ABB RAPID module: Template_20023_Module.mod

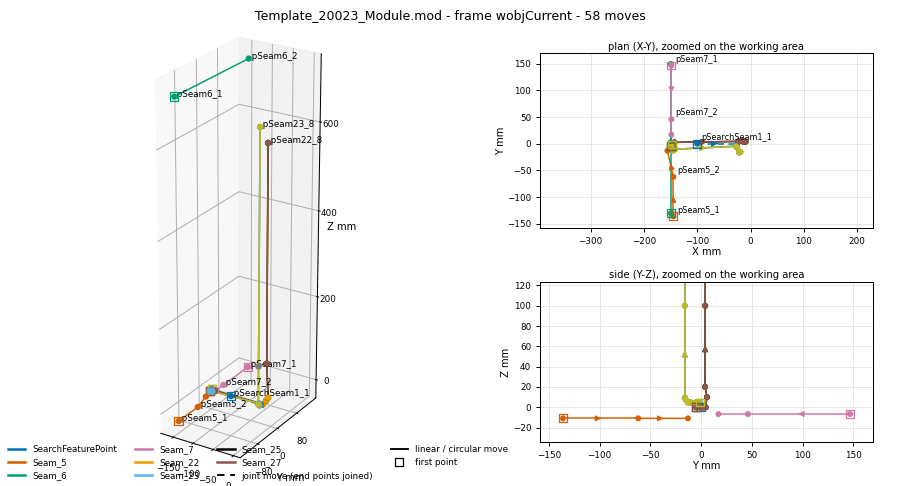
[picture p0: tool path of Template_20023_Module.mod in frame wobjCurrent, 58 of 171 moves have a stored position in this frame; points joined in program order, loops and branches not executed]
MODULE Template_20023_Module
    !*****************************************************
    !Module Name:   Template_20023_Module
    !Version:       1.0
    !Description:   All the targets are coordinated in its self coordinate system
    !Date:          2021-8-21
    !Author:        Michael
    !*****************************************************

    LOCAL PERS num numPartCount:=7;

    !For oframe searching
    LOCAL PERS robtarget pQ1_X1:=[[-75,0,0],[0.37941,0.915976,0.0499502,0.12059],[-1,-1,0,1],[-800,500,456,9E+9,9E+9,9E+9]];
    LOCAL PERS robtarget pQ1_X2:=[[-30,0,0],[0.37941,0.915976,0.0499502,0.12059],[-1,-1,0,1],[-800,500,456,9E+9,9E+9,9E+9]];
    LOCAL PERS robtarget pQ1_Y1:=[[0,75,0],[0.183013,-0.612372,0.683013,-0.353553],[-1,0,-1,1],[-800,500,456,9E+9,9E+9,9E+9]];
    LOCAL PERS robtarget pQ1_Y2:=[[0,200,0],[0.183013,-0.612372,0.683013,-0.353553],[-1,0,-1,1],[-800,500,456,9E+9,9E+9,9E+9]];
    LOCAL PERS robtarget pQ1_Z1:=[[0,0,50],[0.562422,0.303603,0.732963,-0.232963],[-1,-2,-1,1],[-800,500,456,9E+9,9E+9,9E+9]];
    LOCAL PERS robtarget pQ1_Z2:=[[0,0,250],[0.232963,0.732963,-0.303603,0.562422],[-2,-1,1,1],[-800,500,456,9E+9,9E+9,9E+9]];
    LOCAL PERS robtarget pQ1_X1_Found:=[[-75,0,0],[0.37941,0.915976,0.0499502,0.12059],[-1,-1,0,1],[-800,500,456,9E+9,9E+9,9E+9]];
    LOCAL PERS robtarget pQ1_X2_Found:=[[-30,0,0],[0.37941,0.915976,0.0499502,0.12059],[-1,-1,0,1],[-800,500,456,9E+9,9E+9,9E+9]];
    LOCAL PERS robtarget pQ1_Y1_Found:=[[0,75,0],[0.183013,-0.612372,0.683013,-0.353553],[-1,0,-1,1],[-800,500,456,9E+9,9E+9,9E+9]];
    LOCAL PERS robtarget pQ1_Y2_Found:=[[0,200,0],[0.183013,-0.612372,0.683013,-0.353553],[-1,0,-1,1],[-800,500,456,9E+9,9E+9,9E+9]];
    LOCAL PERS robtarget pQ1_Z1_Found:=[[0,0,50],[0.562422,0.303603,0.732963,-0.232963],[-1,-2,-1,1],[-800,500,456,9E+9,9E+9,9E+9]];
    LOCAL PERS robtarget pQ1_Z2_Found:=[[0,0,250],[0.232963,0.732963,-0.303603,0.562422],[-2,-1,1,1],[-800,500,456,9E+9,9E+9,9E+9]];

    LOCAL PERS robtarget pQ2_X1:=[[-75,0,0],[0.37941,0.915976,0.0499502,0.12059],[-1,-1,0,1],[-800,500,456,9E+9,9E+9,9E+9]];
    LOCAL PERS robtarget pQ2_X2:=[[-30,0,0],[0.37941,0.915976,0.0499502,0.12059],[-1,-1,0,1],[-800,500,456,9E+9,9E+9,9E+9]];
    LOCAL PERS robtarget pQ2_Y1:=[[-0.03,74.99,-0.03],[0.0903086,-0.672569,0.657682,-0.327031],[-1,-1,0,1],[-800,500,456.001,9E+09,9E+09,9E+09]];
    LOCAL PERS robtarget pQ2_Y2:=[[-0.03,200,-0.03],[0.0903092,-0.67257,0.657681,-0.327031],[-1,-1,0,1],[-800,500,456.001,9E+09,9E+09,9E+09]];
    LOCAL PERS robtarget pQ2_Z1:=[[0,0,50],[0.562422,0.303603,0.732963,-0.232963],[-1,-2,-1,1],[-800,500,456,9E+9,9E+9,9E+9]];
    LOCAL PERS robtarget pQ2_Z2:=[[0,0,250],[0.232963,0.732963,-0.303603,0.562422],[-2,-1,1,1],[-800,500,456,9E+9,9E+9,9E+9]];
    LOCAL PERS robtarget pQ2_X1_Found:=[[-75,0,0],[0.37941,0.915976,0.0499502,0.12059],[-1,-1,0,1],[-800,500,456,9E+9,9E+9,9E+9]];
    LOCAL PERS robtarget pQ2_X2_Found:=[[-30,0,0],[0.37941,0.915976,0.0499502,0.12059],[-1,-1,0,1],[-800,500,456,9E+9,9E+9,9E+9]];
    LOCAL PERS robtarget pQ2_Y1_Found:=[[17.85,90.22,0.26],[0.183013,-0.612372,0.683013,-0.353553],[-1,0,-1,1],[-800,500,456,9E+09,9E+09,9E+09]];
    LOCAL PERS robtarget pQ2_Y2_Found:=[[14.86,215.24,-0.11],[0.183013,-0.612372,0.683013,-0.353553],[-1,0,-1,1],[-800,500,456,9E+09,9E+09,9E+09]];
    LOCAL PERS robtarget pQ2_Z1_Found:=[[0,0,50],[0.562422,0.303603,0.732963,-0.232963],[-1,-2,-1,1],[-800,500,456,9E+9,9E+9,9E+9]];
    LOCAL PERS robtarget pQ2_Z2_Found:=[[16.02,7.07,231.87],[0.232963,0.732963,-0.303603,0.562422],[-2,-1,1,1],[-800,500,456,9E+09,9E+09,9E+09]];

    LOCAL PERS robtarget pQ3_X1:=[[-75,0,0],[0.37941,0.915976,0.0499502,0.12059],[-1,-1,0,1],[-800,500,456,9E+9,9E+9,9E+9]];
    LOCAL PERS robtarget pQ3_X2:=[[-30,0,0],[0.37941,0.915976,0.0499502,0.12059],[-1,-1,0,1],[-800,500,456,9E+9,9E+9,9E+9]];
    LOCAL PERS robtarget pQ3_Y1:=[[0,-300,0],[0.0890947,0.615873,0.708619,0.332599],[-2,0,-1,1],[-800,-500,450.515,9E+09,9E+09,9E+09]];
    LOCAL PERS robtarget pQ3_Y2:=[[0,-100,0],[0.0890967,0.615873,0.708619,0.332599],[-1,0,-2,1],[-800,-500,450.515,9E+09,9E+09,9E+09]];
    LOCAL PERS robtarget pQ3_Z1:=[[0,0,50],[0.562422,0.303603,0.732963,-0.232963],[-1,-2,-1,1],[-800,500,456,9E+9,9E+9,9E+9]];
    LOCAL PERS robtarget pQ3_Z2:=[[0,0,500],[0.326752,-0.683237,-0.28535,-0.587363],[-1,0,-1,1],[-800,-500,450.515,9E+09,9E+09,9E+09]];
    LOCAL PERS robtarget pQ3_X1_Found:=[[-75,0,0],[0.37941,0.915976,0.0499502,0.12059],[-1,-1,0,1],[-800,500,456,9E+9,9E+9,9E+9]];
    LOCAL PERS robtarget pQ3_X2_Found:=[[-30,0,0],[0.37941,0.915976,0.0499502,0.12059],[-1,-1,0,1],[-800,500,456,9E+9,9E+9,9E+9]];
    LOCAL PERS robtarget pQ3_Y1_Found:=[[5.33,-307.13,27.55],[0.183013,-0.612372,0.683013,-0.353553],[-1,0,-1,1],[-800,500,456,9E+09,9E+09,9E+09]];
    LOCAL PERS robtarget pQ3_Y2_Found:=[[4.1,-107.45,27.54],[0.183013,-0.612372,0.683013,-0.353553],[-1,0,-1,1],[-800,500,456,9E+09,9E+09,9E+09]];
    LOCAL PERS robtarget pQ3_Z1_Found:=[[0,0,50],[0.562422,0.303603,0.732963,-0.232963],[-1,-2,-1,1],[-800,500,456,9E+9,9E+9,9E+9]];
    LOCAL PERS robtarget pQ3_Z2_Found:=[[-3.2,-18.41,500.1],[0.232963,0.732963,-0.303603,0.562422],[-2,-1,1,1],[-800,500,456,9E+09,9E+09,9E+09]];

    LOCAL PERS robtarget pQ4_X1:=[[-75,0,0],[0.37941,0.915976,0.0499502,0.12059],[-1,-1,0,1],[-800,500,456,9E+9,9E+9,9E+9]];
    LOCAL PERS robtarget pQ4_X2:=[[-30,0,0],[0.37941,0.915976,0.0499502,0.12059],[-1,-1,0,1],[-800,500,456,9E+9,9E+9,9E+9]];
    LOCAL PERS robtarget pQ4_Y1:=[[0,75,0],[0.183013,-0.612372,0.683013,-0.353553],[-1,0,-1,1],[-800,500,456,9E+9,9E+9,9E+9]];
    LOCAL PERS robtarget pQ4_Y2:=[[0,200,0],[0.183013,-0.612372,0.683013,-0.353553],[-1,0,-1,1],[-800,500,456,9E+9,9E+9,9E+9]];
    LOCAL PERS robtarget pQ4_Z1:=[[0,0,50],[0.562422,0.303603,0.732963,-0.232963],[-1,-2,-1,1],[-800,500,456,9E+9,9E+9,9E+9]];
    LOCAL PERS robtarget pQ4_Z2:=[[0,0,250],[0.232963,0.732963,-0.303603,0.562422],[-2,-1,1,1],[-800,500,456,9E+9,9E+9,9E+9]];
    LOCAL PERS robtarget pQ4_X1_Found:=[[-75,0,0],[0.37941,0.915976,0.0499502,0.12059],[-1,-1,0,1],[-800,500,456,9E+9,9E+9,9E+9]];
    LOCAL PERS robtarget pQ4_X2_Found:=[[-30,0,0],[0.37941,0.915976,0.0499502,0.12059],[-1,-1,0,1],[-800,500,456,9E+9,9E+9,9E+9]];
    LOCAL PERS robtarget pQ4_Y1_Found:=[[0,75,0],[0.183013,-0.612372,0.683013,-0.353553],[-1,0,-1,1],[-800,500,456,9E+9,9E+9,9E+9]];
    LOCAL PERS robtarget pQ4_Y2_Found:=[[0,200,0],[0.183013,-0.612372,0.683013,-0.353553],[-1,0,-1,1],[-800,500,456,9E+9,9E+9,9E+9]];
    LOCAL PERS robtarget pQ4_Z1_Found:=[[0,0,50],[0.562422,0.303603,0.732963,-0.232963],[-1,-2,-1,1],[-800,500,456,9E+9,9E+9,9E+9]];
    LOCAL PERS robtarget pQ4_Z2_Found:=[[0,0,250],[0.232963,0.732963,-0.303603,0.562422],[-2,-1,1,1],[-800,500,456,9E+9,9E+9,9E+9]];

    LOCAL PERS wobjdata wobjLast:=[FALSE,TRUE,"",[[-455,0,60],[1,0,0,0]],[[3.55142,-18.3921,27.5355],[1,0,0,0]]];
    LOCAL PERS pose poseFrame:=[[3.55142,-18.3921,27.5355],[0.502018,0.494872,0.497955,0.505095]];
    LOCAL PERS pose poseTransform:=[[0,0,0],[0.5,-0.5,-0.5,-0.5]];
    LOCAL PERS pose poseTransform_Q1:=[[0,0,0],[0.5,-0.5,-0.5,-0.5]];
    LOCAL PERS pose poseTransform_Q2:=[[0,0,0],[0.5,-0.5,-0.5,-0.5]];
    LOCAL PERS pose poseTransform_Q3:=[[0,0,0],[0.5,-0.5,-0.5,-0.5]];
    LOCAL PERS pose poseTransform_Q4:=[[0,0,0],[0.5,-0.5,-0.5,-0.5]];

    LOCAL PERS robtarget pSearchSeam1_1:=[[-100,0,0],[0.37941,0.915976,0.0499502,0.12059],[-1,-1,0,1],[-800,500,300,9E+09,9E+09,9E+09]];
    LOCAL PERS robtarget pSearchSeam1_2:=[[-25,0,0],[0.37941,0.915976,0.0499502,0.12059],[-1,-1,0,1],[-800,500,300,9E+09,9E+09,9E+09]];
    LOCAL PERS robtarget pSearchSeam2_1:=[[0,0,50],[0.562422,0.303603,0.732963,-0.232963],[-1,-2,-1,1],[-800,500,456,9E+09,9E+09,9E+09]];
    LOCAL PERS robtarget pSearchSeam2_2:=[[0,0,400],[0.232963,0.732963,-0.303603,0.562422],[-2,-1,1,1],[-800,500,456,9E+09,9E+09,9E+09]];
    LOCAL PERS robtarget pSearchSeam3_1:=[[-100,0,0],[0.260212,-0.95439,0.00662898,-0.146237],[-2,0,0,1],[-772.01,-462.973,258.768,9E+09,9E+09,9E+09]];
    LOCAL PERS robtarget pSearchSeam3_2:=[[-25,0,0],[0.260213,-0.95439,0.00662908,-0.146236],[-2,0,0,1],[-772.01,-462.973,258.768,9E+09,9E+09,9E+09]];
    LOCAL PERS robtarget pSearchSeam4_1:=[[0,0,100],[0.579883,-0.251955,0.739786,0.230156],[-1,1,-4,1],[-843.059,-440.815,465.229,9E+09,9E+09,9E+09]];
    LOCAL PERS robtarget pSearchSeam4_2:=[[0.00,0.00,500.00],[0.243457,-0.745392,-0.234844,-0.574428],[-1,1,-2,1],[-843.059,-440.815,185.21,9E+09,9E+09,9E+09]];
    LOCAL PERS robtarget pSearchSeam5_1:=[[-143.5,-120,0],[0.051556,-0.666714,-0.684628,-0.290031],[-2,0,-1,1],[-800,-500,456,9E+09,9E+09,9E+09]];
    LOCAL PERS robtarget pSearchSeam5_2:=[[-143.5,-50,0],[0.0515572,-0.666714,-0.684629,-0.290031],[-2,0,-1,1],[-800,-500,456,9E+09,9E+09,9E+09]];
    LOCAL PERS robtarget pSearchSeam6_1:=[[-177.86,-120.61,654.68],[1.72416E-05,-0.702562,-0.711622,6.74779E-05],[-2,-1,-2,1],[-529.872,-183.238,-440.181,9E+09,9E+09,9E+09]];
    LOCAL PERS robtarget pSearchSeam6_2:=[[-177.86,122.25,654.68],[1.55975E-05,-0.702564,-0.71162,6.58224E-05],[-2,-1,-2,1],[-529.872,59.6217,-440.181,9E+09,9E+09,9E+09]];
    LOCAL PERS robtarget pSearchSeam7_1:=[[-156.78,138.57,1.27],[0.011391,0.681242,-0.666782,0.301962],[-1,-1,0,1],[-800,500,456.001,9E+09,9E+09,9E+09]];
    LOCAL PERS robtarget pSearchSeam7_2:=[[-156.77,48.60,1.27],[0.0113887,0.681242,-0.666783,0.301962],[-1,-1,0,1],[-800,500.001,456.001,9E+09,9E+09,9E+09]];

    LOCAL PERS robtarget pSeamFound1_1:=[[-105.58,13.08,11.73],[0.37941,0.915976,0.0499502,0.12059],[-1,-1,0,1],[-800,500,456,9E+09,9E+09,9E+09]];
    LOCAL PERS robtarget pSeamFound1_2:=[[-30.16,10.51,12.47],[0.37941,0.915976,0.0499502,0.12059],[-1,-1,0,1],[-800,500,456,9E+09,9E+09,9E+09]];
    LOCAL PERS robtarget pSeamFound2_1:=[[4.12,15.67,52.48],[0.562422,0.303603,0.732963,-0.232963],[-1,-2,-1,1],[-800,500,456,9E+09,9E+09,9E+09]];
    LOCAL PERS robtarget pSeamFound2_2:=[[-7.36,14.86,403.14],[0.232963,0.732963,-0.303603,0.562422],[-2,-1,1,1],[-800,500,456,9E+09,9E+09,9E+09]];
    LOCAL PERS robtarget pSeamFound3_1:=[[-103.01,-4.94,6.01],[0.37941,-0.915976,0.0499502,-0.12059],[-1,0,-1,1],[-800,-500,456,9E+09,9E+09,9E+09]];
    LOCAL PERS robtarget pSeamFound3_2:=[[-28.13,-4.73,6.42],[0.37941,-0.915976,0.0499502,-0.12059],[-1,0,-1,1],[-800,-500,456,9E+09,9E+09,9E+09]];
    LOCAL PERS robtarget pSeamFound4_1:=[[-2.06,0.68,101.12],[0.528109,-0.308093,0.759593,0.221807],[-2,0,0,1],[-800,-500,456,9E+09,9E+09,9E+09]];
    LOCAL PERS robtarget pSeamFound4_2:=[[-4.07,0.38,499.98],[0.232963,-0.732963,-0.303603,-0.562422],[-1,1,-2,1],[-800,-500,456,9E+09,9E+09,9E+09]];
    LOCAL PERS robtarget pSeamFound5_1:=[[-143.5,-119.23,-3.41],[0.183013,0.612372,0.683013,0.353553],[-2,-1,-1,1],[-800,-500,456,9E+09,9E+09,9E+09]];
    LOCAL PERS robtarget pSeamFound5_2:=[[-143.26,-49.3,-3.19],[0.0515551,-0.666714,-0.684629,-0.290031],[-2,0,-1,1],[-800,-500,456,9E+09,9E+09,9E+09]];
    LOCAL PERS robtarget pSeamFound6_1:=[[-167.28,-120.89,729.18],[0.353553,0.683013,0.612372,0.183013],[-1,0,2,1],[-800,500,0,9E+09,9E+09,9E+09]];
    LOCAL PERS robtarget pSeamFound6_2:=[[-165.5,122.06,729.54],[0.353553,0.683013,0.612372,0.183013],[-1,0,2,1],[-800,500,0,9E+09,9E+09,9E+09]];
    LOCAL PERS robtarget pSeamFound7_1:=[[-145.34,136.97,-2.9],[0.183013,-0.612372,0.683013,-0.353553],[-1,0,0,1],[-800,500,456,9E+09,9E+09,9E+09]];
    LOCAL PERS robtarget pSeamFound7_2:=[[-145.37,47.38,-2.17],[0.183013,-0.612372,0.683013,-0.353553],[-1,0,0,1],[-800,500,456,9E+09,9E+09,9E+09]];

    LOCAL PERS robtarget pSeam1_1:=[[-132,0,0],[0.12059,-0.0499502,0.915976,-0.37941],[-1,0,0,1],[-800,500,456,9E+9,9E+9,9E+9]];
    LOCAL PERS robtarget pSeam1_2:=[[-10,0,0],[0.12059,-0.0499502,0.915976,-0.37941],[-1,0,0,1],[-800,500,456,9E+9,9E+9,9E+9]];
    LOCAL PERS robtarget pSeam2_1:=[[0,0,10],[0.232962913,0.732962913,-0.303603179,0.562422224],[-1,-1,0,1],[-800.000011921,500,480.000019073,9E+09,9E+09,9E+09]];
    LOCAL PERS robtarget pSeam2_2:=[[0.00,0.00,100.00],[0.319156,0.553743,-0.253295,0.726188],[-1,-2,1,1],[-800,500,480,9E+09,9E+09,9E+09]];
    LOCAL PERS robtarget pSeam2_3:=[[0,0,385],[0.325934,0.549781,-0.262196,0.723022],[-1,-2,1,1],[-800,500,280,9E+09,9E+09,9E+09]];
    LOCAL PERS robtarget pSeam3_1:=[[-132,-11,0],[0.169082,-0.0700359,0.914659,0.360423],[-2,1,1,1],[-800,-500,456,9E+9,9E+9,9E+9]];
    LOCAL PERS robtarget pSeam3_2:=[[-10,-11,0],[0.169082,-0.0700359,0.914659,0.360423],[-2,1,1,1],[-800,-500,456,9E+9,9E+9,9E+9]];
    LOCAL PERS robtarget pSeam4_1:=[[0.00,-11.00,10.00],[0.266412,-0.657996,-0.396353,-0.582212],[-2,0,2,1],[-800,-500,456,9E+09,9E+09,9E+09]];
    LOCAL PERS robtarget pSeam4_2:=[[0.00,-11.02,99.95],[0.287699,-0.546881,-0.304884,-0.724704],[-2,1,2,1],[-800,-500,456.003,9E+09,9E+09,9E+09]];
    LOCAL PERS robtarget pSeam4_3:=[[0,-11,390],[0.303603,-0.562422,-0.232963,-0.732963],[-2,0,3,1],[-800,-500,256,9E+09,9E+09,9E+09]];
    LOCAL PERS robtarget pSeam5_1:=[[-144.81,-136.21,-10.92],[0.294912,-0.702887,0.64396,-0.0655127],[-1,0,-4,1],[-936.547,-455.411,577.519,9E+09,9E+09,9E+09]];
    LOCAL PERS robtarget pSeam5_2:=[[-144.81,-62.06,-10.92],[0.294912,-0.702886,0.643961,-0.0655098],[-1,0,-4,1],[-936.547,-455.411,577.519,9E+09,9E+09,9E+09]];
    LOCAL PERS robtarget pSeam5_3:=[[-155.95,-13.09,-10.93],[0.326666,-0.70446,0.628926,0.0384397],[-1,0,-4,1],[-760.258,-455.411,577.519,9E+09,9E+09,9E+09]];
    LOCAL PERS robtarget pSeam6_1:=[[-149.47,-130.45,714.57],[0.155044,-0.58872,0.752527,-0.251143],[-1,0,-4,1],[-926.584,-259.409,-310.78,9E+09,9E+09,9E+09]];
    LOCAL PERS robtarget pSeam6_2:=[[-149.47,149.58,711.80],[0.155044,-0.588719,0.752528,-0.251142],[-2,-1,-3,1],[-926.584,-259.408,-310.78,9E+09,9E+09,9E+09]];
    LOCAL PERS robtarget pSeam7_1:=[[-148.49,146.64,-6.67],[0.283896,0.749291,0.591155,0.0922052],[-2,-1,-1,1],[-800,500,456.001,9E+09,9E+09,9E+09]];
    LOCAL PERS robtarget pSeam7_2:=[[-148.49,45.97,-6.67],[0.283895,0.749291,0.591156,0.0922039],[-1,-1,-1,1],[-800,500.001,456.001,9E+09,9E+09,9E+09]];
    LOCAL PERS robtarget pSeam7_3:=[[-148.49,16.98,-6.67],[0.303246,0.758109,0.575904,0.0405837],[-1,-1,-1,1],[-800,500,456.001,9E+09,9E+09,9E+09]];
    LOCAL PERS robtarget pSeam8_1:=[[-144.81,-136.21,-10.92],[0.294912,-0.702887,0.64396,-0.0655127],[-1,0,-4,1],[-936.547,-455.411,577.519,9E+09,9E+09,9E+09]];
    LOCAL PERS robtarget pSeam8_2:=[[-144.81,-62.06,-10.92],[0.294912,-0.702886,0.643961,-0.0655098],[-1,0,-4,1],[-936.547,-455.411,577.519,9E+09,9E+09,9E+09]];
    LOCAL PERS robtarget pSeam8_3:=[[-155.95,-13.09,-10.93],[0.326666,-0.70446,0.628926,0.0384397],[-1,0,-4,1],[-760.258,-455.411,577.519,9E+09,9E+09,9E+09]];
    LOCAL PERS robtarget pSeam9_1:=[[-149.47,-130.45,714.57],[0.155044,-0.58872,0.752527,-0.251143],[-1,0,-4,1],[-926.584,-259.409,-310.78,9E+09,9E+09,9E+09]];
    LOCAL PERS robtarget pSeam9_2:=[[-149.47,149.58,711.8],[0.155044,-0.588719,0.752528,-0.251142],[-2,-1,-3,1],[-926.584,-259.408,-310.78,9E+09,9E+09,9E+09]];
    LOCAL PERS robtarget pSeam10_1:=[[-148.49,146.64,-6.67],[0.283896,0.749291,0.591155,0.0922052],[-2,-1,-1,1],[-800,500,456.001,9E+09,9E+09,9E+09]];
    LOCAL PERS robtarget pSeam10_2:=[[-148.49,45.97,-6.67],[0.283895,0.749291,0.591156,0.0922039],[-1,-1,-1,1],[-800,500.001,456.001,9E+09,9E+09,9E+09]];
    LOCAL PERS robtarget pSeam10_3:=[[-148.49,16.98,-6.67],[0.303246,0.758109,0.575904,0.0405837],[-1,-1,-1,1],[-800,500,456.001,9E+09,9E+09,9E+09]];
    LOCAL PERS robtarget pSeam11_1:=[[-144.81,-136.21,-10.92],[0.294912,-0.702887,0.64396,-0.0655127],[-1,0,-4,1],[-936.547,-455.411,577.519,9E+09,9E+09,9E+09]];
    LOCAL PERS robtarget pSeam11_2:=[[-144.81,-62.06,-10.92],[0.294912,-0.702886,0.643961,-0.0655098],[-1,0,-4,1],[-936.547,-455.411,577.519,9E+09,9E+09,9E+09]];
    LOCAL PERS robtarget pSeam11_3:=[[-155.95,-13.09,-10.93],[0.326666,-0.70446,0.628926,0.0384397],[-1,0,-4,1],[-760.258,-455.411,577.519,9E+09,9E+09,9E+09]];
    LOCAL PERS robtarget pSeam12_1:=[[-149.47,-130.45,714.57],[0.155044,-0.58872,0.752527,-0.251143],[-1,0,-4,1],[-926.584,-259.409,-310.78,9E+09,9E+09,9E+09]];
    LOCAL PERS robtarget pSeam12_2:=[[-149.47,149.58,711.8],[0.155044,-0.588719,0.752528,-0.251142],[-2,-1,-3,1],[-926.584,-259.408,-310.78,9E+09,9E+09,9E+09]];
    LOCAL PERS robtarget pSeam13_1:=[[-148.49,146.64,-6.67],[0.283896,0.749291,0.591155,0.0922052],[-2,-1,-1,1],[-800,500,456.001,9E+09,9E+09,9E+09]];
    LOCAL PERS robtarget pSeam13_2:=[[-148.49,45.97,-6.67],[0.283895,0.749291,0.591156,0.0922039],[-1,-1,-1,1],[-800,500.001,456.001,9E+09,9E+09,9E+09]];
    LOCAL PERS robtarget pSeam13_3:=[[-148.49,16.98,-6.67],[0.303246,0.758109,0.575904,0.0405837],[-1,-1,-1,1],[-800,500,456.001,9E+09,9E+09,9E+09]];
    LOCAL PERS robtarget pSeam14_1:=[[-144.81,-136.21,-10.92],[0.294912,-0.702887,0.64396,-0.0655127],[-1,0,-4,1],[-936.547,-455.411,577.519,9E+09,9E+09,9E+09]];
    LOCAL PERS robtarget pSeam14_2:=[[-144.81,-62.06,-10.92],[0.294912,-0.702886,0.643961,-0.0655098],[-1,0,-4,1],[-936.547,-455.411,577.519,9E+09,9E+09,9E+09]];
    LOCAL PERS robtarget pSeam14_3:=[[-155.95,-13.09,-10.93],[0.326666,-0.70446,0.628926,0.0384397],[-1,0,-4,1],[-760.258,-455.411,577.519,9E+09,9E+09,9E+09]];
    LOCAL PERS robtarget pSeam15_1:=[[-149.47,-130.45,714.57],[0.155044,-0.58872,0.752527,-0.251143],[-1,0,-4,1],[-926.584,-259.409,-310.78,9E+09,9E+09,9E+09]];
    LOCAL PERS robtarget pSeam15_2:=[[-149.47,149.58,711.8],[0.155044,-0.588719,0.752528,-0.251142],[-2,-1,-3,1],[-926.584,-259.408,-310.78,9E+09,9E+09,9E+09]];
    LOCAL PERS robtarget pSeam16_1:=[[-148.49,146.64,-6.67],[0.283896,0.749291,0.591155,0.0922052],[-2,-1,-1,1],[-800,500,456.001,9E+09,9E+09,9E+09]];
    LOCAL PERS robtarget pSeam16_2:=[[-148.49,45.97,-6.67],[0.283895,0.749291,0.591156,0.0922039],[-1,-1,-1,1],[-800,500.001,456.001,9E+09,9E+09,9E+09]];
    LOCAL PERS robtarget pSeam16_3:=[[-148.49,16.98,-6.67],[0.303246,0.758109,0.575904,0.0405837],[-1,-1,-1,1],[-800,500,456.001,9E+09,9E+09,9E+09]];

    LOCAL PERS robtarget pSeam22_1:=[[-150,-4.77,0],[0.147388,0.013946,0.943852,-0.29534],[-1,0,0,1],[-698.527,504.221,467.895,9E+09,9E+09,9E+09]];
    LOCAL PERS robtarget pSeam22_2:=[[-150,1.58,0],[0.147395,0.0139495,0.94385,-0.295344],[-1,0,0,1],[-698.531,504.222,467.895,9E+09,9E+09,9E+09]];
    LOCAL PERS robtarget pSeam22_3:=[[-142.77,2.55,0],[0.147393,0.0139474,0.94385,-0.295343],[-1,0,0,1],[-698.53,504.221,467.894,9E+09,9E+09,9E+09]];
    LOCAL PERS robtarget pSeam22_4:=[[-22.40,4.37,0],[0.261771,-0.0223631,0.919965,-0.29093],[-1,1,0,1],[-698.53,504.221,467.894,9E+09,9E+09,9E+09]];
    LOCAL PERS robtarget pSeam22_5:=[[-15.56,5.63,10],[0.110216,-0.383059,0.740522,-0.54106],[-1,1,-1,1],[-698.53,504.222,467.896,9E+09,9E+09,9E+09]];
    LOCAL PERS robtarget pSeam22_6:=[[-9.32,3.83,20],[0.337928,0.738102,-0.198901,0.549043],[-1,-1,0,1],[-698.53,504.222,467.894,9E+09,9E+09,9E+09]];
    LOCAL PERS robtarget pSeam22_7:=[[-12.94,3.92,100],[0.360942,0.648816,-0.14361,0.65432],[-1,-2,1,1],[-698.53,504.222,467.894,9E+09,9E+09,9E+09]];
    LOCAL PERS robtarget pSeam22_8:=[[-12.93,3.93,599.99],[0.380908,0.526496,-0.160444,0.742946],[-1,-2,1,1],[-698.53,504.225,150.002,9E+09,9E+09,9E+09]];
    LOCAL PERS robtarget pSeam23_1:=[[-147.94,-1.49,4.7],[0.0656464,0.206294,0.89886,0.381031],[-2,-1,-1,1],[-632.83,-462.628,567.927,9E+09,9E+09,9E+09]];
    LOCAL PERS robtarget pSeam23_2:=[[-145.78,-13.08,4.7],[0.0656434,0.206294,0.89886,0.381031],[-2,-1,-1,1],[-632.84,-462.628,567.927,9E+09,9E+09,9E+09]];
    LOCAL PERS robtarget pSeam23_3:=[[-141.46,-10.22,4.7],[0.0656457,0.20629,0.898861,0.38103],[-2,-1,-3,1],[-632.829,-462.628,567.927,9E+09,9E+09,9E+09]];
    LOCAL PERS robtarget pSeam23_4:=[[-27.11,-4.74,5.13],[0.0656436,0.206293,0.89886,0.381032],[-2,-1,-2,1],[-632.84,-462.628,567.927,9E+09,9E+09,9E+09]];
    LOCAL PERS robtarget pSeam23_5:=[[-19.04,-15.21,7.34],[0.155413,-0.57093,-0.596735,-0.542027],[-2,0,-3,1],[-632.84,-462.628,567.927,9E+09,9E+09,9E+09]];
    LOCAL PERS robtarget pSeam23_6:=[[-21.13,-16.17,9.48],[0.307446,-0.708011,-0.25177,-0.583789],[-2,0,-1,1],[-632.84,-462.628,567.927,9E+09,9E+09,9E+09]];
    LOCAL PERS robtarget pSeam23_7:=[[-21.14,-16.17,100.00],[0.357301,-0.602855,-0.220163,-0.67855],[-2,1,-2,1],[-632.84,-462.628,567.927,9E+09,9E+09,9E+09]];
    LOCAL PERS robtarget pSeam23_8:=[[-25.1,-7.29,635.57],[0.358487,-0.433448,-0.169949,-0.809152],[-2,1,-2,1],[-632.84,-462.628,374.549,9E+09,9E+09,9E+09]];

    LOCAL PERS robtarget pSeam25_1:=[[-150,-4.77,0],[0.147388,0.013946,0.943852,-0.29534],[-1,0,0,1],[-698.527,504.221,467.895,9E+09,9E+09,9E+09]];
    LOCAL PERS robtarget pSeam25_2:=[[-150,1.58,0],[0.147395,0.0139495,0.94385,-0.295344],[-1,0,0,1],[-698.531,504.222,467.895,9E+09,9E+09,9E+09]];
    LOCAL PERS robtarget pSeam25_3:=[[-142.77,2.55,0],[0.147393,0.0139474,0.94385,-0.295343],[-1,0,0,1],[-698.53,504.221,467.894,9E+09,9E+09,9E+09]];
    LOCAL PERS robtarget pSeam25_4:=[[-22.40,4.37,0],[0.261771,-0.0223631,0.919965,-0.29093],[-1,1,0,1],[-698.53,504.221,467.894,9E+09,9E+09,9E+09]];
    LOCAL PERS robtarget pSeam25_5:=[[-15.56,5.63,10],[0.110216,-0.383059,0.740522,-0.54106],[-1,1,-1,1],[-698.53,504.222,467.896,9E+09,9E+09,9E+09]];
    LOCAL PERS robtarget pSeam25_6:=[[-9.32,3.83,20],[0.337928,0.738102,-0.198901,0.549043],[-1,-1,0,1],[-698.53,504.222,467.894,9E+09,9E+09,9E+09]];
    LOCAL PERS robtarget pSeam25_7:=[[-12.94,3.92,100],[0.360942,0.648816,-0.14361,0.65432],[-1,-2,1,1],[-698.53,504.222,467.894,9E+09,9E+09,9E+09]];
    LOCAL PERS robtarget pSeam25_8:=[[-12.93,3.93,599.99],[0.380908,0.526496,-0.160444,0.742946],[-1,-2,1,1],[-698.53,504.225,150.002,9E+09,9E+09,9E+09]];
    LOCAL PERS robtarget pSeam26_1:=[[-147.94,-1.49,4.7],[0.0656464,0.206294,0.89886,0.381031],[-2,-1,-1,1],[-632.83,-462.628,567.927,9E+09,9E+09,9E+09]];
    LOCAL PERS robtarget pSeam26_2:=[[-145.78,-13.08,4.7],[0.0656434,0.206294,0.89886,0.381031],[-2,-1,-1,1],[-632.84,-462.628,567.927,9E+09,9E+09,9E+09]];
    LOCAL PERS robtarget pSeam26_3:=[[-141.46,-10.22,4.7],[0.0656457,0.20629,0.898861,0.38103],[-2,-1,-3,1],[-632.829,-462.628,567.927,9E+09,9E+09,9E+09]];
    LOCAL PERS robtarget pSeam26_4:=[[-27.11,-4.74,5.13],[0.0656436,0.206293,0.89886,0.381032],[-2,-1,-2,1],[-632.84,-462.628,567.927,9E+09,9E+09,9E+09]];
    LOCAL PERS robtarget pSeam26_5:=[[-19.04,-15.21,7.34],[0.155413,-0.57093,-0.596735,-0.542027],[-2,0,-3,1],[-632.84,-462.628,567.927,9E+09,9E+09,9E+09]];
    LOCAL PERS robtarget pSeam26_6:=[[-21.13,-16.17,9.48],[0.307446,-0.708011,-0.25177,-0.583789],[-2,0,-1,1],[-632.84,-462.628,567.927,9E+09,9E+09,9E+09]];
    LOCAL PERS robtarget pSeam26_7:=[[-21.14,-16.17,100.00],[0.357301,-0.602855,-0.220163,-0.67855],[-2,1,-2,1],[-632.84,-462.628,567.927,9E+09,9E+09,9E+09]];
    LOCAL PERS robtarget pSeam26_8:=[[-25.1,-7.29,635.57],[0.358487,-0.433448,-0.169949,-0.809152],[-2,1,-2,1],[-632.84,-462.628,374.549,9E+09,9E+09,9E+09]];

    LOCAL PERS robtarget pSeam27_1:=[[-150,-4.77,0],[0.147388,0.013946,0.943852,-0.29534],[-1,0,0,1],[-698.527,504.221,467.895,9E+09,9E+09,9E+09]];
    LOCAL PERS robtarget pSeam27_2:=[[-150,1.58,0],[0.147395,0.0139495,0.94385,-0.295344],[-1,0,0,1],[-698.531,504.222,467.895,9E+09,9E+09,9E+09]];
    LOCAL PERS robtarget pSeam27_3:=[[-142.77,2.55,0],[0.147393,0.0139474,0.94385,-0.295343],[-1,0,0,1],[-698.53,504.221,467.894,9E+09,9E+09,9E+09]];
    LOCAL PERS robtarget pSeam27_4:=[[-22.40,4.37,0],[0.261771,-0.0223631,0.919965,-0.29093],[-1,1,0,1],[-698.53,504.221,467.894,9E+09,9E+09,9E+09]];
    LOCAL PERS robtarget pSeam27_5:=[[-15.56,5.63,10],[0.110216,-0.383059,0.740522,-0.54106],[-1,1,-1,1],[-698.53,504.222,467.896,9E+09,9E+09,9E+09]];
    LOCAL PERS robtarget pSeam27_6:=[[-9.32,3.83,20],[0.337928,0.738102,-0.198901,0.549043],[-1,-1,0,1],[-698.53,504.222,467.894,9E+09,9E+09,9E+09]];
    LOCAL PERS robtarget pSeam27_7:=[[-12.94,3.92,100],[0.360942,0.648816,-0.14361,0.65432],[-1,-2,1,1],[-698.53,504.222,467.894,9E+09,9E+09,9E+09]];
    LOCAL PERS robtarget pSeam27_8:=[[-12.93,3.93,599.99],[0.380908,0.526496,-0.160444,0.742946],[-1,-2,1,1],[-698.53,504.225,150.002,9E+09,9E+09,9E+09]];
    LOCAL PERS robtarget pSeam28_1:=[[-147.94,-1.49,4.7],[0.0656464,0.206294,0.89886,0.381031],[-2,-1,-1,1],[-632.83,-462.628,567.927,9E+09,9E+09,9E+09]];
    LOCAL PERS robtarget pSeam28_2:=[[-145.78,-13.08,4.7],[0.0656434,0.206294,0.89886,0.381031],[-2,-1,-1,1],[-632.84,-462.628,567.927,9E+09,9E+09,9E+09]];
    LOCAL PERS robtarget pSeam28_3:=[[-141.46,-10.22,4.7],[0.0656457,0.20629,0.898861,0.38103],[-2,-1,-3,1],[-632.829,-462.628,567.927,9E+09,9E+09,9E+09]];
    LOCAL PERS robtarget pSeam28_4:=[[-27.11,-4.74,5.13],[0.0656436,0.206293,0.89886,0.381032],[-2,-1,-2,1],[-632.84,-462.628,567.927,9E+09,9E+09,9E+09]];
    LOCAL PERS robtarget pSeam28_5:=[[-19.04,-15.21,7.34],[0.155413,-0.57093,-0.596735,-0.542027],[-2,0,-3,1],[-632.84,-462.628,567.927,9E+09,9E+09,9E+09]];
    LOCAL PERS robtarget pSeam28_6:=[[-21.13,-16.17,9.48],[0.307446,-0.708011,-0.25177,-0.583789],[-2,0,-1,1],[-632.84,-462.628,567.927,9E+09,9E+09,9E+09]];
    LOCAL PERS robtarget pSeam28_7:=[[-21.14,-16.17,100.00],[0.357301,-0.602855,-0.220163,-0.67855],[-2,1,-2,1],[-632.84,-462.628,567.927,9E+09,9E+09,9E+09]];
    LOCAL PERS robtarget pSeam28_8:=[[-25.1,-7.29,635.57],[0.358487,-0.433448,-0.169949,-0.809152],[-2,1,-2,1],[-632.84,-462.628,374.549,9E+09,9E+09,9E+09]];

    !Only used to compensate Absolute Accuracy Offset
    LOCAL PERS pos posAOSeam1_1:=[0,0,0];
    LOCAL PERS pos posAOSeam1_2:=[0,0,0];
    LOCAL PERS pos posAOSeam2_1:=[0,-2,0];
    LOCAL PERS pos posAOSeam2_2:=[0,-2,0];
    LOCAL PERS pos posAOSeam2_3:=[6,0,0];
    LOCAL PERS pos posAOSeam3_1:=[4,0,-6];
    LOCAL PERS pos posAOSeam3_2:=[0,-6,0];
    LOCAL PERS pos posAOSeam4_1:=[-2,3,0];
    LOCAL PERS pos posAOSeam4_2:=[-1,6,0];
    LOCAL PERS pos posAOSeam4_3:=[0,10,0];
    LOCAL PERS pos posAOSeam5_1:=[0,0,0];
    LOCAL PERS pos posAOSeam5_2:=[0,0,0];
    LOCAL PERS pos posAOSeam5_3:=[0,0,0];
    LOCAL PERS pos posAOSeam6_1:=[17,0,-15];
    LOCAL PERS pos posAOSeam6_2:=[17,0,-15];
    LOCAL PERS pos posAOSeam7_1:=[-2,0,0];
    LOCAL PERS pos posAOSeam7_2:=[-2,0,0];
    LOCAL PERS pos posAOSeam7_3:=[-2,0,0];
    LOCAL PERS pos posAOSeam8_1:=[0,0,0];
    LOCAL PERS pos posAOSeam8_2:=[0,0,0];
    LOCAL PERS pos posAOSeam8_3:=[0,0,0];
    LOCAL PERS pos posAOSeam9_1:=[-20,0,0];
    LOCAL PERS pos posAOSeam9_2:=[-20,0,0];
    LOCAL PERS pos posAOSeam10_1:=[0,0,0];
    LOCAL PERS pos posAOSeam10_2:=[0,0,0];
    LOCAL PERS pos posAOSeam10_3:=[0,0,0];
    LOCAL PERS pos posAOSeam11_1:=[-16,-4,-25];
    LOCAL PERS pos posAOSeam11_2:=[-16,-4,-25];
    LOCAL PERS pos posAOSeam11_3:=[-16,0,-25];
    LOCAL PERS pos posAOSeam12_1:=[-15,-23,-10];
    LOCAL PERS pos posAOSeam12_2:=[-15,-23,-10];
    LOCAL PERS pos posAOSeam13_1:=[-3,-14,-15];
    LOCAL PERS pos posAOSeam13_2:=[-3,-15,-18];
    LOCAL PERS pos posAOSeam13_3:=[-3,-15,-15];
    LOCAL PERS pos posAOSeam14_1:=[-16,-4,-25];
    LOCAL PERS pos posAOSeam14_2:=[-16,-4,-25];
    LOCAL PERS pos posAOSeam14_3:=[-16,0,-25];
    LOCAL PERS pos posAOSeam15_1:=[-15,-23,-10];
    LOCAL PERS pos posAOSeam15_2:=[-15,-23,-10];
    LOCAL PERS pos posAOSeam16_1:=[-3,-14,-15];
    LOCAL PERS pos posAOSeam16_2:=[-3,-15,-18];
    LOCAL PERS pos posAOSeam16_3:=[-3,-15,-15];

    LOCAL PERS pos posAOSeam22_1:=[15,0,-15];
    LOCAL PERS pos posAOSeam22_2:=[17,-1,-15];
    LOCAL PERS pos posAOSeam22_3:=[12,-2,-15];
    LOCAL PERS pos posAOSeam22_4:=[-20,3,-12];
    LOCAL PERS pos posAOSeam22_5:=[-12,1,-3];
    LOCAL PERS pos posAOSeam22_6:=[-6,0,10];
    LOCAL PERS pos posAOSeam22_7:=[-3,-3,0];
    LOCAL PERS pos posAOSeam22_8:=[3,3,50];
    LOCAL PERS pos posAOSeam23_1:=[2,0,-20];
    LOCAL PERS pos posAOSeam23_2:=[2,-1,-20];
    LOCAL PERS pos posAOSeam23_3:=[3,0,-20];
    LOCAL PERS pos posAOSeam23_4:=[-22,0,-15];
    LOCAL PERS pos posAOSeam23_5:=[-17,8,-7];
    LOCAL PERS pos posAOSeam23_6:=[-13,8,0];
    LOCAL PERS pos posAOSeam23_7:=[-13,0,0];
    LOCAL PERS pos posAOSeam23_8:=[-14,0,0];

    LOCAL PERS pos posAOSeam25_1:=[15,0,-15];
    LOCAL PERS pos posAOSeam25_2:=[17,-1,-15];
    LOCAL PERS pos posAOSeam25_3:=[12,-2,-15];
    LOCAL PERS pos posAOSeam25_4:=[-20,-6,-12];
    LOCAL PERS pos posAOSeam25_5:=[-12,-5,-6];
    LOCAL PERS pos posAOSeam25_6:=[-2,-4,5];
    LOCAL PERS pos posAOSeam25_7:=[0,-3,0];
    LOCAL PERS pos posAOSeam25_8:=[5,1,50];
    LOCAL PERS pos posAOSeam26_1:=[2,0,-23];
    LOCAL PERS pos posAOSeam26_2:=[2,-1,-24];
    LOCAL PERS pos posAOSeam26_3:=[3,0,-22];
    LOCAL PERS pos posAOSeam26_4:=[-22,0,-15];
    LOCAL PERS pos posAOSeam26_5:=[-17,8,-7];
    LOCAL PERS pos posAOSeam26_6:=[-13,8,0];
    LOCAL PERS pos posAOSeam26_7:=[-13,6,0];
    LOCAL PERS pos posAOSeam26_8:=[-14,7,0];

    LOCAL PERS pos posAOSeam27_1:=[15,0,-15];
    LOCAL PERS pos posAOSeam27_2:=[17,-1,-15];
    LOCAL PERS pos posAOSeam27_3:=[12,-2,-15];
    LOCAL PERS pos posAOSeam27_4:=[-20,-6,-12];
    LOCAL PERS pos posAOSeam27_5:=[-12,-5,-6];
    LOCAL PERS pos posAOSeam27_6:=[-2,-4,5];
    LOCAL PERS pos posAOSeam27_7:=[0,-3,0];
    LOCAL PERS pos posAOSeam27_8:=[5,1,50];
    LOCAL PERS pos posAOSeam28_1:=[2,0,-23];
    LOCAL PERS pos posAOSeam28_2:=[2,-1,-24];
    LOCAL PERS pos posAOSeam28_3:=[3,0,-22];
    LOCAL PERS pos posAOSeam28_4:=[-22,0,-15];
    LOCAL PERS pos posAOSeam28_5:=[-17,8,-7];
    LOCAL PERS pos posAOSeam28_6:=[-13,8,0];
    LOCAL PERS pos posAOSeam28_7:=[-13,6,0];
    LOCAL PERS pos posAOSeam28_8:=[-14,7,0];

    !Used for PDispSet
    LOCAL PERS pose peSeam1_1:=[[0.155304,-6.36427,1.11146],[1,0,0,0]];
    LOCAL PERS pose peSeam1_2:=[[0.0753555,-3.29217,1.66705],[1,0,0,0]];
    LOCAL PERS pose peSeam2_1:=[[0.607692,-1.74091,0.0125351],[1,0,0,0]];
    LOCAL PERS pose peSeam2_2:=[[-1.0559,-2.19269,-0.0204926],[1,0,0,0]];
    LOCAL PERS pose peSeam2_3:=[[-0.32395,-1.62331,-0.125092],[1,0,0,0]];
    LOCAL PERS pose peSeam3_1:=[[4.12688,-4.41331,-8.79105],[1,0,0,0]];
    LOCAL PERS pose peSeam3_2:=[[0.0145874,-6.72514,-3.08223],[1,0,0,0]];
    LOCAL PERS pose peSeam4_1:=[[-8.09118,3.01741,-0.0262299],[1,0,0,0]];
    LOCAL PERS pose peSeam4_2:=[[-7.48061,5.27455,-0.0342102],[1,0,0,0]];
    LOCAL PERS pose peSeam4_3:=[[-7.73635,6.79469,-0.0606995],[1,0,0,0]];
    LOCAL PERS pose peSeam5_1:=[[1.25163,-0.0277557,7.45649],[1,0,0,0]];
    LOCAL PERS pose peSeam5_2:=[[1.5061,-0.0293579,7.68976],[1,0,0,0]];
    LOCAL PERS pose peSeam5_3:=[[12.814,-0.0686913,7.8537],[1,0,0,0]];
    LOCAL PERS pose peSeam6_1:=[[-0.879242,0.10936,-0.403992],[1,0,0,0]];
    LOCAL PERS pose peSeam6_2:=[[1.17229,0.0896301,2.78088],[1,0,0,0]];
    LOCAL PERS pose peSeam7_1:=[[1.15326,0.0290222,3.69097],[1,0,0,0]];
    LOCAL PERS pose peSeam7_2:=[[1.11955,0.0357208,4.5112],[1,0,0,0]];
    LOCAL PERS pose peSeam7_3:=[[1.10985,0.0376396,4.7474],[1,0,0,0]];
    LOCAL PERS pose peSeam8_1:=[[2.8342,0.0904541,-4.80138],[1,0,0,0]];
    LOCAL PERS pose peSeam8_2:=[[-0.692978,0.00148392,-4.16271],[1,0,0,0]];
    LOCAL PERS pose peSeam8_3:=[[-0.692978,0.00148392,-4.16271],[1,0,0,0]];
    LOCAL PERS pose peSeam9_1:=[[-22.565,0.286362,30.3056],[1,0,0,0]];
    LOCAL PERS pose peSeam9_2:=[[-28.5206,0.127365,27.0722],[1,0,0,0]];
    LOCAL PERS pose peSeam10_1:=[[1.15506,0.0231094,-0.816231],[1,0,0,0]];
    LOCAL PERS pose peSeam10_2:=[[-0.668945,-0.010788,-0.566907],[1,0,0,0]];
    LOCAL PERS pose peSeam10_3:=[[-0.668945,-0.010788,-0.566907],[1,0,0,0]];
    LOCAL PERS pose peSeam11_1:=[[2.49045,-3.97635,-1.28609],[1,0,0,0]];
    LOCAL PERS pose peSeam11_2:=[[2.3,-3.9767,-1.248],[1,0,0,0]];
    LOCAL PERS pose peSeam11_3:=[[2.23366,0.0231609,-1.18673],[1,0,0,0]];
    LOCAL PERS pose peSeam12_1:=[[6.03051,-22.3034,23.6097],[1,0,0,0]];
    LOCAL PERS pose peSeam12_2:=[[6.63764,-22.2961,22.8259],[1,0,0,0]];
    LOCAL PERS pose peSeam13_1:=[[-10.9162,-13.8462,2.57889],[1,0,0,0]];
    LOCAL PERS pose peSeam13_2:=[[-8.08952,-14.7266,1.79651],[1,0,0,0]];
    LOCAL PERS pose peSeam13_3:=[[-7.20422,-14.6892,5.49105],[1,0,0,0]];
    LOCAL PERS pose peSeam14_1:=[[2.49045,-3.97635,-1.28609],[1,0,0,0]];
    LOCAL PERS pose peSeam14_2:=[[2.3,-3.9767,-1.248],[1,0,0,0]];
    LOCAL PERS pose peSeam14_3:=[[2.23366,0.0231609,-1.18673],[1,0,0,0]];
    LOCAL PERS pose peSeam15_1:=[[6.03051,-22.3034,23.6097],[1,0,0,0]];
    LOCAL PERS pose peSeam15_2:=[[6.63764,-22.2961,22.8259],[1,0,0,0]];
    LOCAL PERS pose peSeam16_1:=[[-10.9162,-13.8462,2.57889],[1,0,0,0]];
    LOCAL PERS pose peSeam16_2:=[[-8.08952,-14.7266,1.79651],[1,0,0,0]];
    LOCAL PERS pose peSeam16_3:=[[-7.20422,-14.6892,5.49105],[1,0,0,0]];

    LOCAL PERS pose peSeam22_1:=[[15.5483,19.345,-3.70046],[1,0,0,0]];
    LOCAL PERS pose peSeam22_2:=[[17.3322,12.0023,-3.70258],[1,0,0,0]];
    LOCAL PERS pose peSeam22_3:=[[12.2901,9.78739,-3.63205],[1,0,0,0]];
    LOCAL PERS pose peSeam22_4:=[[8.20701,8.87295,0.546895],[1,0,0,0]];
    LOCAL PERS pose peSeam22_5:=[[9.0474,5.37828,-0.385536],[1,0,0,0]];
    LOCAL PERS pose peSeam22_6:=[[8.48691,5.96049,2.67717],[1,0,0,0]];
    LOCAL PERS pose peSeam22_7:=[[12.4868,8.639,0.533897],[1,0,0,0]];
    LOCAL PERS pose peSeam22_8:=[[2.12562,13.4753,49.9955],[1,0,0,0]];
    LOCAL PERS pose peSeam23_1:=[[2.0042,-3.57599,-18.936],[1,0,0,0]];
    LOCAL PERS pose peSeam23_2:=[[1.97162,7.01997,-18.9243],[1,0,0,0]];
    LOCAL PERS pose peSeam23_3:=[[2.97948,5.17211,-18.9006],[1,0,0,0]];
    LOCAL PERS pose peSeam23_4:=[[3.53306,0.0128403,-13.7045],[1,0,0,0]];
    LOCAL PERS pose peSeam23_5:=[[0.452089,18.5054,-7.87036],[1,0,0,0]];
    LOCAL PERS pose peSeam23_6:=[[6.53125,19.4596,-3.02176],[1,0,0,0]];
    LOCAL PERS pose peSeam23_7:=[[6.08509,16.8508,0.108849],[1,0,0,0]];
    LOCAL PERS pose peSeam23_8:=[[6.34617,7.56794,0.108276],[1,0,0,0]];

    LOCAL PERS pose peSeam25_1:=[[15.5483,19.345,-3.70046],[1,0,0,0]];
    LOCAL PERS pose peSeam25_2:=[[17.3322,12.0023,-3.70258],[1,0,0,0]];
    LOCAL PERS pose peSeam25_3:=[[12.2901,9.78739,-3.63205],[1,0,0,0]];
    LOCAL PERS pose peSeam25_4:=[[8.20701,8.87295,0.546895],[1,0,0,0]];
    LOCAL PERS pose peSeam25_5:=[[9.0474,5.37828,-0.385536],[1,0,0,0]];
    LOCAL PERS pose peSeam25_6:=[[8.48691,5.96049,2.67717],[1,0,0,0]];
    LOCAL PERS pose peSeam25_7:=[[12.4868,8.639,0.533897],[1,0,0,0]];
    LOCAL PERS pose peSeam25_8:=[[2.12562,13.4753,49.9955],[1,0,0,0]];
    LOCAL PERS pose peSeam26_1:=[[2.0042,-3.57599,-18.936],[1,0,0,0]];
    LOCAL PERS pose peSeam26_2:=[[1.97162,7.01997,-18.9243],[1,0,0,0]];
    LOCAL PERS pose peSeam26_3:=[[2.97948,5.17211,-18.9006],[1,0,0,0]];
    LOCAL PERS pose peSeam26_4:=[[3.53306,0.0128403,-13.7045],[1,0,0,0]];
    LOCAL PERS pose peSeam26_5:=[[0.452089,18.5054,-7.87036],[1,0,0,0]];
    LOCAL PERS pose peSeam26_6:=[[6.53125,19.4596,-3.02176],[1,0,0,0]];
    LOCAL PERS pose peSeam26_7:=[[6.08509,16.8508,0.108849],[1,0,0,0]];
    LOCAL PERS pose peSeam26_8:=[[6.34617,7.56794,0.108276],[1,0,0,0]];

    LOCAL PERS pose peSeam27_1:=[[15.5483,19.345,-3.70046],[1,0,0,0]];
    LOCAL PERS pose peSeam27_2:=[[17.3322,12.0023,-3.70258],[1,0,0,0]];
    LOCAL PERS pose peSeam27_3:=[[12.2901,9.78739,-3.63205],[1,0,0,0]];
    LOCAL PERS pose peSeam27_4:=[[8.20701,8.87295,0.546895],[1,0,0,0]];
    LOCAL PERS pose peSeam27_5:=[[9.0474,5.37828,-0.385536],[1,0,0,0]];
    LOCAL PERS pose peSeam27_6:=[[8.48691,5.96049,2.67717],[1,0,0,0]];
    LOCAL PERS pose peSeam27_7:=[[12.4868,8.639,0.533897],[1,0,0,0]];
    LOCAL PERS pose peSeam27_8:=[[2.12562,13.4753,49.9955],[1,0,0,0]];
    LOCAL PERS pose peSeam28_1:=[[2.0042,-3.57599,-18.936],[1,0,0,0]];
    LOCAL PERS pose peSeam28_2:=[[1.97162,7.01997,-18.9243],[1,0,0,0]];
    LOCAL PERS pose peSeam28_3:=[[2.97948,5.17211,-18.9006],[1,0,0,0]];
    LOCAL PERS pose peSeam28_4:=[[3.53306,0.0128403,-13.7045],[1,0,0,0]];
    LOCAL PERS pose peSeam28_5:=[[0.452089,18.5054,-7.87036],[1,0,0,0]];
    LOCAL PERS pose peSeam28_6:=[[6.53125,19.4596,-3.02176],[1,0,0,0]];
    LOCAL PERS pose peSeam28_7:=[[6.08509,16.8508,0.108849],[1,0,0,0]];
    LOCAL PERS pose peSeam28_8:=[[6.34617,7.56794,0.108276],[1,0,0,0]];

    !Only for local welding parameters
    LOCAL PERS welddata weld_1:=[6,0,[38,0,-1,0,0,350,0,0,0],[0,0,0,0,0,0,0,0,0]];
    LOCAL PERS weavedata weave_1:=[1,0,4,6,0,0,0,0,0,0,0,0,0,0,0];
    LOCAL PERS trackdata track_1:=[0,TRUE,50,[0,30,30,0,0,0,0,0,0],[0,0,0,0,0,0,0]];

    !wobjCurrent must be set correctly
    !extOffsetCurrent must be set correctly
    PROC Template_20023()
        Logging "Start to run Template_20023...";
        SetGO Go112_WeldCompleted,0;
        SetGO Go80_WeldingStatus,0;

        IF boolEnableGantryOffset THEN
            LoadGantryOffset;
        ENDIF

        MoveToReadyQuadrant 3;
        IF boolEnableSearch THEN
            SearchAndProcess;
        ENDIF

        WeldSeam 23;
        MoveToReadyQuadrant 3;

        MoveToReadyQuadrant 2;
        WeldSeam 22;
        WeldSeam 7;
        MoveToReadyQuadrant 2;

        MoveToReadyQuadrant 3;
        WeldSeam 6;
        WeldSeam 5;
        WeldSeam 25;
        MoveToReadyQuadrant 3;

        MoveToReadyQuadrant 2;
        WeldSeam 26;
        WeldSeam 10;
        MoveToReadyQuadrant 2;

        MoveToReadyQuadrant 3;
        WeldSeam 9;
        WeldSeam 8;
        WeldSeam 27;
        MoveToReadyQuadrant 3;

        MoveToReadyQuadrant 2;
        WeldSeam 28;
        WeldSeam 13;
        MoveToReadyQuadrant 2;

        MoveToReadyQuadrant 3;
        WeldSeam 12;
        WeldSeam 11;
        MoveToReadyQuadrant 3;

        MoveToReadyQuadrant 2;
        WeldSeam 16;
        MoveToReadyQuadrant 2;

        MoveToReadyQuadrant 3;
        WeldSeam 15;
        WeldSeam 14;
        MoveToReadyQuadrant 3;


        EOffsOff;
        Incr numPartCount;
        Logging "Template_20023 is done";

    UNDO
        EOffsOff;
    ENDPROC

    !1 - Search the fine oframe
    !2 - Search the seam offset if needed
    LOCAL PROC SearchAndProcess()
        SearchOframe;
        !SearchFeaturePoint;
        !ProcessFeaturePoint;
    ENDPROC

    LOCAL PROC SearchFeaturePoint()
        Logging "SearchFeaturePoint";
        MoveAbsJ [[-0.442793,-43.1611,0,20,-65.6482,0],[-500,500,0,9E+09,9E+09,9E+09]],speedAir,fine,toolLaser\WObj:=wobjCurrent;
        MoveJ pSearchSeam1_1,speedAproach,fine,toolLaser\WObj:=wobjCurrent;
        MoveJ pSearchSeam1_2,speedAproach,fine,toolLaser\WObj:=wobjCurrent;
    ENDPROC

    LOCAL PROC ProcessFeaturePoint()
        Logging "ProcessFeaturePoint";
        pSeam1_1.trans.y:=pSearchSeam1_1.trans.y;
        pSeam1_1.trans.z:=pSearchSeam1_1.trans.z;
        pSeam1_2.trans.y:=pSearchSeam1_2.trans.y;
        pSeam1_2.trans.z:=pSearchSeam1_2.trans.z;

    ENDPROC

    LOCAL PROC SearchOframe()
        Logging "Search oframe";
        wobjCurrent.oframe:=[[0,0,0],[1,0,0,0]];

        MoveAbsJ [[-69.8437,-39.8871,45.8877,34.3389,-62.4823,-125.956],[-800,-500,450.515,9E+09,9E+09,9E+09]],speedAir,zoneAir,toolLaser\WObj:=wobjCurrent;
        ScanSeamByLaser pQ3_Y1_Found,pQ3_Y1,scanJoint2,speedAproach,toolLaser\WObj:=wobjCurrent;
        ScanSeamByLaser pQ3_Y2_Found,pQ3_Y2,scanJoint2,speedAproach,toolLaser\WObj:=wobjCurrent;
        MoveAbsJ [[-105.635,-11.9899,28.2629,12.7016,-67.9619,-83.0548],[-800,-500,450.515,9E+09,9E+09,9E+09]],speedAir,zoneAir,toolLaser\WObj:=wobjCurrent;

        !MoveAbsJ [[-89.7306,-43.1368,0,-20,-65.7254,9.9994],[-800,500,0,9E+09,9E+09,9E+09]],speedAir,zoneAir,toolLaser\WObj:=wobjCurrent;
        !ScanSeamByLaser pQ3_X1_Found,pQ3_X1,scanJoint2,speedAproach,toolLaser\WObj:=wobjCurrent;
        !ScanSeamByLaser pQ3_X2_Found,pQ3_X2,scanJoint2,speedAproach,toolLaser\WObj:=wobjCurrent;
        !MoveAbsJ [[-89.7306,-43.1368,0,-20,-65.7254,9.9994],[-800,500,0,9E+09,9E+09,9E+09]],speedAir,zoneAir,toolLaser\WObj:=wobjCurrent;

        !MoveAbsJ [[-92.7971,-23.7414,5.96932,0,-45.8213,6.36111E-15],[-800,500,0,9E+9,9E+9,9E+9]],speedAir,zoneAir,toolLaser\WObj:=wobjCurrent;
        !ScanSeamByLaser pQ3_Z1_Found,pQ3_Z1,scanJoint2,speedAproach,toolLaser\WObj:=wobjCurrent;
        MoveAbsJ [[-59.855,-15.8981,15.8975,84.4084,-81.9376,-82.7938],[-800,-500,450.515,9E+09,9E+09,9E+09]],speedAir,zoneAir,toolLaser\WObj:=wobjCurrent;
        ScanSeamByLaser pQ3_Z2_Found,pQ3_Z2,scanJoint2,speedAproach,toolLaser\WObj:=wobjCurrent;
        MoveAbsJ [[-59.855,-15.8981,15.8975,84.4084,-81.9376,-82.7938],[-800,-500,450.515,9E+09,9E+09,9E+09]],speedAir,zoneAir,toolLaser\WObj:=wobjCurrent;

        !Search YPXN in Wobj0
        poseTransform.rot:=OrientZYX(-90,0,0);
        !Search YPZP in Wobj0
        poseTransform.rot:=OrientZYX(0,-90,-90);

        poseTransform_Q3:=poseTransform;

        poseFrame:=DefFrame(pQ3_Y1_Found,pQ3_Y2_Found,pQ3_Z2_Found\Origin:=3);
        Logging "poseFrame.trans:="+ValToStr(poseFrame.trans);
        Logging "poseFrame.rot:="+GetEulerAngleString(poseFrame.rot);
        wobjCurrent.oframe:=PoseMult(poseFrame,poseTransform);
        !wobjCurrent.oframe.trans:=[0,0,0];
        wobjCurrent.oframe.rot:=[1,0,0,0];
        Logging "oframe.trans:="+ValToStr(wobjCurrent.oframe.trans);
        Logging "oframe.rot:="+GetEulerAngleString(wobjCurrent.oframe.rot);

        wobjLast:=wobjCurrent;
        WriteSysDataLog "Template_20023";

    ENDPROC

    LOCAL PROC CopySeamTargets()
        peSeam25_1:=peSeam22_1;
        peSeam25_2:=peSeam22_2;
        peSeam25_3:=peSeam22_3;
        peSeam25_4:=peSeam22_4;
        peSeam25_5:=peSeam22_5;
        peSeam25_6:=peSeam22_6;
        peSeam25_7:=peSeam22_7;
        peSeam25_8:=peSeam22_8;
        peSeam26_1:=peSeam23_1;
        peSeam26_2:=peSeam23_2;
        peSeam26_3:=peSeam23_3;
        peSeam26_4:=peSeam23_4;
        peSeam26_5:=peSeam23_5;
        peSeam26_6:=peSeam23_6;
        peSeam26_7:=peSeam23_7;
        peSeam26_8:=peSeam23_8;

        peSeam27_1:=peSeam22_1;
        peSeam27_2:=peSeam22_2;
        peSeam27_3:=peSeam22_3;
        peSeam27_4:=peSeam22_4;
        peSeam27_5:=peSeam22_5;
        peSeam27_6:=peSeam22_6;
        peSeam27_7:=peSeam22_7;
        peSeam27_8:=peSeam22_8;
        peSeam28_1:=peSeam23_1;
        peSeam28_2:=peSeam23_2;
        peSeam28_3:=peSeam23_3;
        peSeam28_4:=peSeam23_4;
        peSeam28_5:=peSeam23_5;
        peSeam28_6:=peSeam23_6;
        peSeam28_7:=peSeam23_7;
        peSeam28_8:=peSeam23_8;

        pSeam8_1:=pSeam5_1;
        pSeam8_2:=pSeam5_2;
        pSeam8_3:=pSeam5_3;
        pSeam9_1:=pSeam6_1;
        pSeam9_2:=pSeam6_2;
        pSeam10_1:=pSeam7_1;
        pSeam10_2:=pSeam7_2;
        pSeam10_3:=pSeam7_3;

        pSeam11_1:=pSeam5_1;
        pSeam11_2:=pSeam5_2;
        pSeam11_3:=pSeam5_3;
        pSeam12_1:=pSeam6_1;
        pSeam12_2:=pSeam6_2;
        pSeam13_1:=pSeam7_1;
        pSeam13_2:=pSeam7_2;
        pSeam13_3:=pSeam7_3;

        pSeam14_1:=pSeam5_1;
        pSeam14_2:=pSeam5_2;
        pSeam14_3:=pSeam5_3;
        pSeam15_1:=pSeam6_1;
        pSeam15_2:=pSeam6_2;
        pSeam16_1:=pSeam7_1;
        pSeam16_2:=pSeam7_2;
        pSeam16_3:=pSeam7_3;
    ENDPROC

    LOCAL PROC WeldSeam(num numSeamIndex)
        UpdateWeldSeamStatus\Start,numSeamIndex;
        %"Seam_"+ValToStr(numSeamIndex)%;
        UpdateWeldSeamStatus numSeamIndex;
    ENDPROC

    LOCAL PROC Seam_5()
        MoveAbsJ [[-90,-45.3776,29.7093,-26.0507,-60,-89.658],[-800.001,-500,1.11759E-05,9E+09,9E+09,9E+09]],speedAir,zoneAir,toolLaser\WObj:=wobjCurrent;
        ScanSeamByLaser pSeamFound5_1,pSearchSeam5_1,scanJoint5,speedAproach,toolLaser\WObj:=wobjCurrent;
        ScanSeamByLaser pSeamFound5_2,pSearchSeam5_2,scanJoint5,speedAproach,toolLaser\WObj:=wobjCurrent;
        MoveAbsJ [[-85.4494,-0.322939,17.5128,29.3144,-80.8065,-182.429],[-993.313,-551.941,314.402,9E+09,9E+09,9E+09]],speedAir,zoneAir,toolLaser\WObj:=wobjCurrent;

        MoveAbsJ [[-67.412,14.846,-0.645323,49.0808,-93.8906,-295.656],[-1229.43,-453.211,577.519,9E+09,9E+09,9E+09]],speedAir,zoneAir,toolWeldGun\WObj:=wobjCurrent;

        RefreshDisp\X\Y\Z,peSeam5_1,posAOSeam5_1,pSeam5_1,pSeamFound5_1,pSeamFound5_2;
        MoveJ GetAproachTarget(pSeam5_1),speedAir,zoneAir,toolWeldGun\WObj:=wobjCurrent;
        ArcLStart pSeam5_1,speedAproach,seamShared,weldShared_3\Weave:=weaveShared_3,fine,toolWeldGun\WObj:=wobjCurrent\Track:=trackShared_3\SeamName:="WeldSeam";
        RefreshDisp\X\Y\Z,peSeam5_2,posAOSeam5_2,pSeam5_2,pSeamFound5_1,pSeamFound5_2;
        ArcL pSeam5_2,speedWeld,seamShared,weldShared_3\Weave:=weaveShared_3,zoneWeld,toolWeldGun\WObj:=wobjCurrent\Track:=trackShared_3;
        RefreshDisp\X\Y\Z,peSeam5_3,posAOSeam5_3,pSeam5_3,pSeamFound5_1,pSeamFound5_2;
        ArcLEnd pSeam5_3,speedWeld,seamShared,weldShared_3\Weave:=weaveShared_3,fine,toolWeldGun\WObj:=wobjCurrent\Track:=trackShared_3;
        MoveL GetAproachTarget(pSeam5_2),speedAir,zoneAir,toolWeldGun\WObj:=wobjCurrent;
        PDispOff;

        MoveAbsJ [[-51.1655,-13.5142,1.89254,52.2752,-74.0337,-289.751],[-1112.37,-455.41,-93.8066,9E+09,9E+09,9E+09]],speedAir,zoneAir,toolWeldGun\WObj:=wobjCurrent;

    UNDO
        PDispOff;
    ENDPROC

    LOCAL PROC Seam_6()
        MoveAbsJ [[-90.5701,-15.1713,15.5771,-0.00383681,-90.4126,-90.1633],[-696.437,-431.442,-440.181,9E+09,9E+09,9E+09]],speedAir,zoneAir,toolLaser\WObj:=wobjCurrent;
        ScanSeamByLaser pSeamFound6_1,pSearchSeam6_1,scanJoint9,speedAproach,toolLaser\WObj:=wobjCurrent;
        ScanSeamByLaser pSeamFound6_2,pSearchSeam6_2,scanJoint9,speedAproach,toolLaser\WObj:=wobjCurrent;
        MoveAbsJ [[-90.5717,-15.1715,15.5768,-0.933082,-47.2982,-180.511],[-1165.55,-259.408,-427.247,9E+09,9E+09,9E+09]],speedAir,zoneAir,toolLaser\WObj:=wobjCurrent;

        MoveAbsJ [[-90.5717,-15.1678,15.9076,-0.928039,-47.6325,-260.567],[-1023.24,-259.408,-310.78,9E+09,9E+09,9E+09]],speedAir,zoneAir,toolWeldGun\WObj:=wobjCurrent;

        RefreshDisp\X\Y\Z,peSeam6_1,posAOSeam6_1,pSeam6_1,pSeamFound6_1,pSeamFound6_2;
        MoveJ GetAproachTarget(pSeam6_1),speedAir,zoneAir,toolWeldGun\WObj:=wobjCurrent;
        ArcLStart pSeam6_1,speedAproach,seamShared,weldShared_3\Weave:=weaveShared_3,fine,toolWeldGun\WObj:=wobjCurrent\Track:=trackShared_3\SeamName:="WeldSeam";
        RefreshDisp\X\Y\Z,peSeam6_2,posAOSeam6_2,pSeam6_2,pSeamFound6_1,pSeamFound6_2;
        ArcLEnd pSeam6_2,speedWeld,seamShared,weldShared_3\Weave:=weaveShared_3,fine,toolWeldGun\WObj:=wobjCurrent\Track:=trackShared_3;
        MoveL GetAproachTarget(pSeam6_2),speedAir,zoneAir,toolWeldGun\WObj:=wobjCurrent;
        PDispOff;

        MoveAbsJ [[-117.562,12.6034,16.1097,-6.52503,-81.3331,-236.497],[-1141.85,-489.878,-310.78,9E+09,9E+09,9E+09]],speedAir,zoneAir,toolWeldGun\WObj:=wobjCurrent;

    UNDO
        PDispOff;
    ENDPROC

    LOCAL PROC Seam_7()
        MoveAbsJ [[-46.062,-60,29.8365,31.1131,-33.8128,32.5521],[-800,500,0,9E+09,9E+09,9E+09]],speedAir,zoneAir,toolLaser\WObj:=wobjCurrent;
        ScanSeamByLaser pSeamFound7_1,pSearchSeam7_1,scanJoint7,speedAproach,toolLaser\WObj:=wobjCurrent;
        ScanSeamByLaser pSeamFound7_2,pSearchSeam7_2,scanJoint7,speedAproach,toolLaser\WObj:=wobjCurrent;
        MoveAbsJ [[-46.062,-60,29.8365,31.1131,-33.8128,32.5521],[-800,500,0,9E+9,9E+9,9E+9]],speedAir,zoneAir,toolLaser\WObj:=wobjCurrent;

        MoveAbsJ [[-84.3237,-22.0998,43.9819,-23.3004,-66.6329,-87.802],[-800,500,456.001,9E+09,9E+09,9E+09]],speedAir,zoneAir,toolWeldGun\WObj:=wobjCurrent;

        RefreshDisp\X\Y\Z,peSeam7_1,posAOSeam7_1,pSeam7_1,pSeamFound7_1,pSeamFound7_2;
        MoveJ GetAproachTarget(pSeam7_1),speedAir,zoneAir,toolWeldGun\WObj:=wobjCurrent;
        ArcLStart pSeam7_1,speedAproach,seamShared,weldShared_3\Weave:=weaveShared_3,fine,toolWeldGun\WObj:=wobjCurrent\Track:=trackShared_3\SeamName:="WeldSeam";
        RefreshDisp\X\Y\Z,peSeam7_2,posAOSeam7_2,pSeam7_2,pSeamFound7_1,pSeamFound7_2;
        ArcL pSeam7_2,speedWeld,seamShared,weldShared_3\Weave:=weaveShared_3,zoneWeld,toolWeldGun\WObj:=wobjCurrent\Track:=trackShared_3;
        RefreshDisp\X\Y\Z,peSeam7_3,posAOSeam7_3,pSeam7_3,pSeamFound7_1,pSeamFound7_2;
        ArcLEnd pSeam7_3,speedWeld,seamShared,weldShared_3\Weave:=weaveShared_3,fine,toolWeldGun\WObj:=wobjCurrent\Track:=trackShared_3;
        MoveL GetAproachTarget(pSeam7_2),speedAir,zoneAir,toolWeldGun\WObj:=wobjCurrent;
        PDispOff;

        MoveAbsJ [[-116.79,14.4276,-5.44873,-46.8373,-95.7932,-49.4616],[-800,599.47,59.6006,9E+09,9E+09,9E+09]],speedAir,zoneAir,toolWeldGun\WObj:=wobjCurrent;

    UNDO
        PDispOff;
    ENDPROC

    LOCAL PROC Seam_8()
        MoveAbsJ [[-71.556,-47.9334,28.2436,31.7192,-45.8965,-223.034],[-962.587,-574.971,78.9099,9E+09,9E+09,9E+09]],speedAir,zoneAir,toolWeldGun\WObj:=wobjCurrent;

        RefreshDisp\X\Y\Z,peSeam8_1,posAOSeam8_1,pSeam8_1,pSeamFound5_1,pSeamFound5_2;
        MoveJ GetAproachTarget(pSeam8_1),speedAir,zoneAir,toolWeldGun\WObj:=wobjCurrent;
        ArcLStart pSeam8_1,speedAproach,seamShared,weldShared_3\Weave:=weaveShared_3,fine,toolWeldGun\WObj:=wobjCurrent\Track:=trackShared_3\SeamName:="WeldSeam";
        RefreshDisp\X\Y\Z,peSeam8_2,posAOSeam8_2,pSeam8_2,pSeamFound5_1,pSeamFound5_2;
        ArcL pSeam8_2,speedWeld,seamShared,weldShared_3\Weave:=weaveShared_3,zoneWeld,toolWeldGun\WObj:=wobjCurrent\Track:=trackShared_3;
        RefreshDisp\X\Y\Z,peSeam8_3,posAOSeam8_3,pSeam8_3,pSeamFound5_1,pSeamFound5_2;
        ArcLEnd pSeam8_3,speedWeld,seamShared,weldShared_3\Weave:=weaveShared_3,fine,toolWeldGun\WObj:=wobjCurrent\Track:=trackShared_3;
        MoveL GetAproachTarget(pSeam8_2),speedAir,zoneAir,toolWeldGun\WObj:=wobjCurrent;
        PDispOff;

        MoveAbsJ [[-41.0418,-31.5876,26.0872,55.1135,-96.0722,-271.732],[-1052.23,-501.078,28.2565,9E+09,9E+09,9E+09]],speedAir,zoneAir,toolWeldGun\WObj:=wobjCurrent;

    UNDO
        PDispOff;
    ENDPROC

    LOCAL PROC Seam_9()
        MoveAbsJ [[-33.5777,-14.1948,-7.14305,31.9006,-54.7255,-329.895],[-974.292,26.6024,-153.782,9E+09,9E+09,9E+09]],speedAir,zoneAir,toolWeldGun\WObj:=wobjCurrent;

        RefreshDisp\X\Y\Z,peSeam9_1,posAOSeam9_1,pSeam9_1,pSeamFound6_1,pSeamFound6_2;
        MoveJ GetAproachTarget(pSeam9_1),speedAir,zoneAir,toolWeldGun\WObj:=wobjCurrent;
        ArcLStart pSeam9_1,speedAproach,seamShared,weldShared_3\Weave:=weaveShared_3,fine,toolWeldGun\WObj:=wobjCurrent\Track:=trackShared_3\SeamName:="WeldSeam";
        RefreshDisp\X\Y\Z,peSeam9_2,posAOSeam9_2,pSeam9_2,pSeamFound6_1,pSeamFound6_2;
        ArcLEnd pSeam9_2,speedWeld,seamShared,weldShared_3\Weave:=weaveShared_3,fine,toolWeldGun\WObj:=wobjCurrent\Track:=trackShared_3;
        MoveL GetAproachTarget(pSeam9_2),speedAir,zoneAir,toolWeldGun\WObj:=wobjCurrent;
        PDispOff;

        MoveAbsJ [[-95.2212,-57.4908,23.9722,28.9891,-13.2344,-189.739],[-1030.97,16.5018,-37.1456,9E+09,9E+09,9E+09]],speedAir,zoneAir,toolWeldGun\WObj:=wobjCurrent;

    UNDO
        PDispOff;
    ENDPROC

    LOCAL PROC Seam_10()
        MoveAbsJ [[-57.8525,-46.5622,23.0288,10.0453,-41.145,3.82011],[-800,500,0,9E+09,9E+09,9E+09]],speedAir,zoneAir,toolWeldGun\WObj:=wobjCurrent;

        RefreshDisp\X\Y\Z,peSeam10_1,posAOSeam10_1,pSeam10_1,pSeamFound7_1,pSeamFound7_2;
        MoveJ GetAproachTarget(pSeam10_1),speedAir,zoneAir,toolWeldGun\WObj:=wobjCurrent;
        ArcLStart pSeam10_1,speedAproach,seamShared,weldShared_3\Weave:=weaveShared_3,fine,toolWeldGun\WObj:=wobjCurrent\Track:=trackShared_3\SeamName:="WeldSeam";
        RefreshDisp\X\Y\Z,peSeam10_2,posAOSeam10_2,pSeam10_2,pSeamFound7_1,pSeamFound7_2;
        ArcL pSeam10_2,speedWeld,seamShared,weldShared_3\Weave:=weaveShared_3,zoneWeld,toolWeldGun\WObj:=wobjCurrent\Track:=trackShared_3;
        RefreshDisp\X\Y\Z,peSeam10_3,posAOSeam10_3,pSeam10_3,pSeamFound7_1,pSeamFound7_2;
        ArcLEnd pSeam10_3,speedWeld,seamShared,weldShared_3\Weave:=weaveShared_3,fine,toolWeldGun\WObj:=wobjCurrent\Track:=trackShared_3;
        MoveL GetAproachTarget(pSeam10_2),speedAir,zoneAir,toolWeldGun\WObj:=wobjCurrent;
        PDispOff;

        MoveAbsJ [[-57.8525,-46.5622,23.0288,10.0453,-41.145,3.82011],[-800,500,0,9E+9,9E+9,9E+9]],speedAir,zoneAir,toolWeldGun\WObj:=wobjCurrent;

    UNDO
        PDispOff;
    ENDPROC

    LOCAL PROC Seam_11()
        MoveAbsJ [[-90.0958,-51.82,19.8196,31.233,-19.0313,-205.181],[-1001.63,-502.947,-7.06924,9E+09,9E+09,9E+09]],speedAir,zoneAir,toolWeldGun\WObj:=wobjCurrent;

        RefreshDisp\X\Y\Z,peSeam11_1,posAOSeam11_1,pSeam11_1,pSeamFound5_1,pSeamFound5_2;
        MoveJ GetAproachTarget(pSeam11_1),speedAir,zoneAir,toolWeldGun\WObj:=wobjCurrent;
        ArcLStart pSeam11_1,speedAproach,seamShared,weldShared_3\Weave:=weaveShared_3,fine,toolWeldGun\WObj:=wobjCurrent\Track:=trackShared_3\SeamName:="WeldSeam";
        RefreshDisp\X\Y\Z,peSeam11_2,posAOSeam11_2,pSeam11_2,pSeamFound5_1,pSeamFound5_2;
        ArcL pSeam11_2,speedWeld,seamShared,weldShared_3\Weave:=weaveShared_3,zoneWeld,toolWeldGun\WObj:=wobjCurrent\Track:=trackShared_3;
        RefreshDisp\X\Y\Z,peSeam11_3,posAOSeam11_3,pSeam11_3,pSeamFound5_1,pSeamFound5_2;
        ArcLEnd pSeam11_3,speedWeld,seamShared,weldShared_3\Weave:=weaveShared_3,fine,toolWeldGun\WObj:=wobjCurrent\Track:=trackShared_3;
        MoveL GetAproachTarget(pSeam11_2),speedAir,zoneAir,toolWeldGun\WObj:=wobjCurrent;
        PDispOff;

        MoveAbsJ [[-41.0418,-31.5876,26.0872,55.1135,-96.0722,-271.732],[-1052.23,-501.078,28.2565,9E+09,9E+09,9E+09]],speedAir,zoneAir,toolWeldGun\WObj:=wobjCurrent;

    UNDO
        PDispOff;
    ENDPROC

    LOCAL PROC Seam_12()
        MoveAbsJ [[-33.5777,-14.1948,-7.14305,31.9006,-54.7255,-329.895],[-974.292,26.6024,-153.782,9E+09,9E+09,9E+09]],speedAir,zoneAir,toolWeldGun\WObj:=wobjCurrent;

        RefreshDisp\X\Y\Z,peSeam12_1,posAOSeam12_1,pSeam12_1,pSeamFound6_1,pSeamFound6_2;
        MoveJ GetAproachTarget(pSeam12_1),speedAir,zoneAir,toolWeldGun\WObj:=wobjCurrent;
        ArcLStart pSeam12_1,speedAproach,seamShared,weldShared_3\Weave:=weaveShared_3,fine,toolWeldGun\WObj:=wobjCurrent\Track:=trackShared_3\SeamName:="WeldSeam";
        RefreshDisp\X\Y\Z,peSeam12_2,posAOSeam12_2,pSeam12_2,pSeamFound6_1,pSeamFound6_2;
        ArcLEnd pSeam12_2,speedWeld,seamShared,weldShared_3\Weave:=weaveShared_3,fine,toolWeldGun\WObj:=wobjCurrent\Track:=trackShared_3;
        MoveL GetAproachTarget(pSeam12_2),speedAir,zoneAir,toolWeldGun\WObj:=wobjCurrent;
        PDispOff;

        MoveAbsJ [[-95.2212,-57.4908,23.9722,28.9891,-13.2344,-189.739],[-1030.97,16.5018,-37.1456,9E+09,9E+09,9E+09]],speedAir,zoneAir,toolWeldGun\WObj:=wobjCurrent;

    UNDO
        PDispOff;
    ENDPROC

    LOCAL PROC Seam_13()
        MoveAbsJ [[-57.8525,-46.5622,23.0288,10.0453,-41.145,3.82011],[-800,500,0,9E+09,9E+09,9E+09]],speedAir,zoneAir,toolWeldGun\WObj:=wobjCurrent;

        RefreshDisp\X\Y\Z,peSeam13_1,posAOSeam13_1,pSeam13_1,pSeamFound7_1,pSeamFound7_2;
        MoveJ GetAproachTarget(pSeam13_1),speedAir,zoneAir,toolWeldGun\WObj:=wobjCurrent;
        ArcLStart pSeam13_1,speedAproach,seamShared,weldShared_3\Weave:=weaveShared_3,fine,toolWeldGun\WObj:=wobjCurrent\Track:=trackShared_3\SeamName:="WeldSeam";
        RefreshDisp\X\Y\Z,peSeam13_2,posAOSeam13_2,pSeam13_2,pSeamFound7_1,pSeamFound7_2;
        ArcL pSeam13_2,speedWeld,seamShared,weldShared_3\Weave:=weaveShared_3,zoneWeld,toolWeldGun\WObj:=wobjCurrent\Track:=trackShared_3;
        RefreshDisp\X\Y\Z,peSeam13_3,posAOSeam13_3,pSeam13_3,pSeamFound7_1,pSeamFound7_2;
        ArcLEnd pSeam13_3,speedWeld,seamShared,weldShared_3\Weave:=weaveShared_3,fine,toolWeldGun\WObj:=wobjCurrent\Track:=trackShared_3;
        MoveL GetAproachTarget(pSeam13_2),speedAir,zoneAir,toolWeldGun\WObj:=wobjCurrent;
        PDispOff;

        MoveAbsJ [[-57.8525,-46.5622,23.0288,10.0453,-41.145,3.82011],[-800,500,0,9E+9,9E+9,9E+9]],speedAir,zoneAir,toolWeldGun\WObj:=wobjCurrent;

    UNDO
        PDispOff;
    ENDPROC

    LOCAL PROC Seam_14()
        MoveAbsJ [[-91.7336,-51.0976,19.6248,30.665,-17.9291,-207.595],[-994.15,-506.227,-10.8218,9E+09,9E+09,9E+09]],speedAir,zoneAir,toolWeldGun\WObj:=wobjCurrent;

        RefreshDisp\X\Y\Z,peSeam14_1,posAOSeam14_1,pSeam14_1,pSeamFound5_1,pSeamFound5_2;
        MoveJ GetAproachTarget(pSeam14_1),speedAir,zoneAir,toolWeldGun\WObj:=wobjCurrent;
        ArcLStart pSeam14_1,speedAproach,seamShared,weldShared_3\Weave:=weaveShared_3,fine,toolWeldGun\WObj:=wobjCurrent\Track:=trackShared_3\SeamName:="WeldSeam";
        RefreshDisp\X\Y\Z,peSeam14_2,posAOSeam14_2,pSeam14_2,pSeamFound5_1,pSeamFound5_2;
        ArcL pSeam14_2,speedWeld,seamShared,weldShared_3\Weave:=weaveShared_3,zoneWeld,toolWeldGun\WObj:=wobjCurrent\Track:=trackShared_3;
        RefreshDisp\X\Y\Z,peSeam14_3,posAOSeam14_3,pSeam14_3,pSeamFound5_1,pSeamFound5_2;
        ArcLEnd pSeam14_3,speedWeld,seamShared,weldShared_3\Weave:=weaveShared_3,fine,toolWeldGun\WObj:=wobjCurrent\Track:=trackShared_3;
        MoveL GetAproachTarget(pSeam14_2),speedAir,zoneAir,toolWeldGun\WObj:=wobjCurrent;
        PDispOff;

        MoveAbsJ [[-41.0418,-31.5876,26.0872,55.1135,-96.0722,-271.732],[-1052.23,-501.078,28.2565,9E+09,9E+09,9E+09]],speedAir,zoneAir,toolWeldGun\WObj:=wobjCurrent;

    UNDO
        PDispOff;
    ENDPROC

    LOCAL PROC Seam_15()
        MoveAbsJ [[-33.5777,-14.1948,-7.14305,31.9006,-54.7255,-329.895],[-974.292,26.6024,-153.782,9E+09,9E+09,9E+09]],speedAir,zoneAir,toolWeldGun\WObj:=wobjCurrent;

        RefreshDisp\X\Y\Z,peSeam15_1,posAOSeam15_1,pSeam15_1,pSeamFound6_1,pSeamFound6_2;
        MoveJ GetAproachTarget(pSeam15_1),speedAir,zoneAir,toolWeldGun\WObj:=wobjCurrent;
        ArcLStart pSeam15_1,speedAproach,seamShared,weldShared_3\Weave:=weaveShared_3,fine,toolWeldGun\WObj:=wobjCurrent\Track:=trackShared_3\SeamName:="WeldSeam";
        RefreshDisp\X\Y\Z,peSeam15_2,posAOSeam15_2,pSeam15_2,pSeamFound6_1,pSeamFound6_2;
        ArcLEnd pSeam15_2,speedWeld,seamShared,weldShared_3\Weave:=weaveShared_3,fine,toolWeldGun\WObj:=wobjCurrent\Track:=trackShared_3;
        MoveL GetAproachTarget(pSeam15_2),speedAir,zoneAir,toolWeldGun\WObj:=wobjCurrent;
        PDispOff;

        MoveAbsJ [[-95.2212,-57.4908,23.9722,28.9891,-13.2344,-189.739],[-1030.97,16.5018,-37.1456,9E+09,9E+09,9E+09]],speedAir,zoneAir,toolWeldGun\WObj:=wobjCurrent;

    UNDO
        PDispOff;
    ENDPROC

    LOCAL PROC Seam_16()
        MoveAbsJ [[-57.8525,-46.5622,23.0288,10.0453,-41.145,3.82011],[-800,500,0,9E+09,9E+09,9E+09]],speedAir,zoneAir,toolWeldGun\WObj:=wobjCurrent;

        RefreshDisp\X\Y\Z,peSeam16_1,posAOSeam16_1,pSeam16_1,pSeamFound7_1,pSeamFound7_2;
        MoveJ GetAproachTarget(pSeam16_1),speedAir,zoneAir,toolWeldGun\WObj:=wobjCurrent;
        ArcLStart pSeam16_1,speedAproach,seamShared,weldShared_3\Weave:=weaveShared_3,fine,toolWeldGun\WObj:=wobjCurrent\Track:=trackShared_3\SeamName:="WeldSeam";
        RefreshDisp\X\Y\Z,peSeam16_2,posAOSeam16_2,pSeam16_2,pSeamFound7_1,pSeamFound7_2;
        ArcL pSeam16_2,speedWeld,seamShared,weldShared_3\Weave:=weaveShared_3,zoneWeld,toolWeldGun\WObj:=wobjCurrent\Track:=trackShared_3;
        RefreshDisp\X\Y\Z,peSeam16_3,posAOSeam16_3,pSeam16_3,pSeamFound7_1,pSeamFound7_2;
        ArcLEnd pSeam16_3,speedWeld,seamShared,weldShared_3\Weave:=weaveShared_3,fine,toolWeldGun\WObj:=wobjCurrent\Track:=trackShared_3;
        MoveL GetAproachTarget(pSeam16_2),speedAir,zoneAir,toolWeldGun\WObj:=wobjCurrent;
        PDispOff;

        MoveAbsJ [[-57.8525,-46.5622,23.0288,10.0453,-41.145,3.82011],[-800,500,0,9E+9,9E+9,9E+9]],speedAir,zoneAir,toolWeldGun\WObj:=wobjCurrent;

    UNDO
        PDispOff;
    ENDPROC

    LOCAL PROC Seam_22()
        MoveAbsJ [[-89.7306,-43.1368,0,-20,-65.7254,-90],[-800,500,0,9E+09,9E+09,9E+09]],speedAir,zoneAir,toolLaser\WObj:=wobjCurrent;
        ScanSeamByLaser pSeamFound1_1,pSearchSeam1_1,scanJoint1,speedAproach,toolLaser\WObj:=wobjCurrent;
        ScanSeamByLaser pSeamFound1_2,pSearchSeam1_2,scanJoint1,speedAproach,toolLaser\WObj:=wobjCurrent;
        MoveAbsJ [[-151.286,-18.7531,-14.2564,-45.3536,-84.2743,-60],[-800,500,230.338,9E+09,9E+09,9E+09]],speedAir,zoneAir,toolLaser\WObj:=wobjCurrent;
        ScanSeamByLaser pSeamFound2_1,pSearchSeam2_1,scanJoint2,speedAproach,toolLaser\WObj:=wobjCurrent;
        ScanSeamByLaser pSeamFound2_2,pSearchSeam2_2,scanJoint2,speedAproach,toolLaser\WObj:=wobjCurrent;
        MoveAbsJ [[-91.6084,-32.3753,-0.280293,-50.9631,-57.0723,194.327],[-800,500,207.46,9E+09,9E+09,9E+09]],speedAir,zoneAir,toolLaser\WObj:=wobjCurrent;

        MoveAbsJ [[-52.7557,-43.8883,36.8223,15.4091,-52.0967,115.276],[-737.076,502.617,361.603,9E+09,9E+09,9E+09]],speedAir,zoneAir,toolWeldGun\WObj:=wobjCurrent;

        RefreshDisp\X\Y\Z,peSeam22_1,posAOSeam22_1,pSeam22_1,pSeamFound1_1,pSeamFound1_2;
        MoveJ GetAproachTarget(pSeam22_1),speedAir,zoneAir,toolWeldGun\WObj:=wobjCurrent;
        ArcLStart pSeam22_1,speedAproach,seamShared,weldShared_1\Weave:=weaveShared_1,fine,toolWeldGun\WObj:=wobjCurrent\Track:=trackShared_1\SeamName:="WeldSeam";
        RefreshDisp\X\Y\Z,peSeam22_2,posAOSeam22_2,pSeam22_2,pSeamFound1_1,pSeamFound1_2;
        ArcL pSeam22_2,speedWeld,seamShared,weldShared_1\Weave:=weaveShared_1,zoneWeld,toolWeldGun\WObj:=wobjCurrent\Track:=trackShared_1;
        RefreshDisp\X\Y\Z,peSeam22_3,posAOSeam22_3,pSeam22_3,pSeamFound1_1,pSeamFound1_2;
        ArcL pSeam22_3,speedWeld,seamShared,weldShared_1\Weave:=weaveShared_1,zoneWeld,toolWeldGun\WObj:=wobjCurrent\Track:=trackShared_1;
        RefreshDisp\Y\Z,peSeam22_4,posAOSeam22_4,pSeam22_4,pSeamFound1_1,pSeamFound1_2;
        RefreshDisp\X,peSeam22_4,posAOSeam22_4,pSeam22_4,pSeamFound2_1,pSeamFound2_2;
        ArcL pSeam22_4,speedWeld,seamShared,weldShared_1\Weave:=weaveShared_1,zoneWeld,toolWeldGun\WObj:=wobjCurrent\Track:=trackShared_1;
        RefreshDisp\Y\Z,peSeam22_5,posAOSeam22_5,pSeam22_5,pSeamFound1_1,pSeamFound1_2;
        RefreshDisp\X,peSeam22_5,posAOSeam22_5,pSeam22_5,pSeamFound2_1,pSeamFound2_2;
        ArcL pSeam22_5,speedAproach,seamShared,weldShared_6\Weave:=weaveShared_6,zoneWeld,toolWeldGun\WObj:=wobjCurrent\Track:=trackShared_7;
        RefreshDisp\Y\Z,peSeam22_6,posAOSeam22_6,pSeam22_6,pSeamFound1_1,pSeamFound1_2;
        RefreshDisp\X,peSeam22_6,posAOSeam22_6,pSeam22_6,pSeamFound2_1,pSeamFound2_2;
        ArcL pSeam22_6,speedWeld,seamShared,weldShared_6\Weave:=weaveShared_6,zoneWeld,toolWeldGun\WObj:=wobjCurrent\Track:=trackShared_7;
        RefreshDisp\X\Y\Z,peSeam22_7,posAOSeam22_7,pSeam22_7,pSeamFound2_1,pSeamFound2_2;
        ArcL pSeam22_7,speedWeld,seamShared,weldShared_2\Weave:=weaveShared_2,zoneWeld,toolWeldGun\WObj:=wobjCurrent\Track:=trackShared_2;
        RefreshDisp\X\Y\Z,peSeam22_8,posAOSeam22_8,pSeam22_8,pSeamFound2_1,pSeamFound2_2;
        ArcLEnd pSeam22_8,speedWeld,seamShared,weldShared_2\Weave:=weaveShared_2,fine,toolWeldGun\WObj:=wobjCurrent\Track:=trackShared_2;
        MoveL GetAproachTarget(pSeam22_8),speedAir,zoneAir,toolWeldGun\WObj:=wobjCurrent;
        PDispOff;

        MoveAbsJ [[-94.6272,-62.3288,31.5236,-67.9884,-28.6289,132.373],[-732.484,502.809,100,9E+09,9E+09,9E+09]],speedAir,zoneAir,toolWeldGun\WObj:=wobjCurrent;

    UNDO
        PDispOff;
    ENDPROC

    LOCAL PROC Seam_23()
        !Stop;
        MoveAbsJ [[-86.8272,-23.9992,11.9198,34.1856,-65.0959,-13.587],[-772.01,-462.973,258.768,9E+09,9E+09,9E+09]],speedAir,zoneAir,toolLaser\WObj:=wobjCurrent;
        ScanSeamByLaser pSeamFound3_1,pSearchSeam3_1,scanJoint3,speedAproach,toolLaser\WObj:=wobjCurrent;
        ScanSeamByLaser pSeamFound3_2,pSearchSeam3_2,scanJoint3,speedAproach,toolLaser\WObj:=wobjCurrent;
        MoveAbsJ [[-86.827,-23.9992,11.9199,34.1856,-65.0957,-13.587],[-772.01,-462.974,258.768,9E+09,9E+09,9E+09]],speedAir,zoneAir,toolLaser\WObj:=wobjCurrent;
        ScanSeamByLaser pSeamFound4_1,pSearchSeam4_1,scanJoint4,speedAproach,toolLaser\WObj:=wobjCurrent;
        ScanSeamByLaser pSeamFound4_2,pSearchSeam4_2,scanJoint4,speedAproach,toolLaser\WObj:=wobjCurrent;
        MoveAbsJ [[-80.4049,-44.6685,20.3534,67.5249,-47.9841,-114.985],[-796.262,-445.671,220.606,9E+09,9E+09,9E+09]],speedAir,zoneAir,toolLaser\WObj:=wobjCurrent;

        MoveAbsJ [[-130.927,-60.2857,31.9214,-11.7127,-13.6227,-93.7947],[-632.831,-462.628,344.22,9E+09,9E+09,9E+09]],speedAir,zoneAir,toolWeldGun\WObj:=wobjCurrent;

        RefreshDisp\X\Y\Z,peSeam23_1,posAOSeam23_1,pSeam23_1,pSeamFound3_1,pSeamFound3_2;
        MoveJ GetAproachTarget(pSeam23_1),speedAir,zoneAir,toolWeldGun\WObj:=wobjCurrent;
        ArcLStart pSeam23_1,speedAproach,seamShared,weldShared_1\Weave:=weaveShared_1,fine,toolWeldGun\WObj:=wobjCurrent\Track:=trackShared_1\SeamName:="WeldSeam";
        RefreshDisp\X\Y\Z,peSeam23_2,posAOSeam23_2,pSeam23_2,pSeamFound3_1,pSeamFound3_2;
        ArcL pSeam23_2,speedWeld,seamShared,weldShared_1\Weave:=weaveShared_1,zoneWeld,toolWeldGun\WObj:=wobjCurrent\Track:=trackShared_1;
        RefreshDisp\X\Y\Z,peSeam23_3,posAOSeam23_3,pSeam23_3,pSeamFound3_1,pSeamFound3_2;
        ArcL pSeam23_3,speedWeld,seamShared,weldShared_1\Weave:=weaveShared_1,zoneWeld,toolWeldGun\WObj:=wobjCurrent\Track:=trackShared_1;
        RefreshDisp\Y\Z,peSeam23_4,posAOSeam23_4,pSeam23_4,pSeamFound3_1,pSeamFound3_2;
        RefreshDisp\X,peSeam23_4,posAOSeam23_4,pSeam23_4,pSeamFound4_1,pSeamFound4_2;
        ArcL pSeam23_4,speedWeld,seamShared,weldShared_1\Weave:=weaveShared_1,zoneWeld,toolWeldGun\WObj:=wobjCurrent\Track:=trackShared_1;
        RefreshDisp\Y\Z,peSeam23_5,posAOSeam23_5,pSeam23_5,pSeamFound3_1,pSeamFound3_2;
        RefreshDisp\X,peSeam23_5,posAOSeam23_5,pSeam23_5,pSeamFound4_1,pSeamFound4_2;
        ArcL pSeam23_5,speedAproach,seamShared,weldShared_7\Weave:=weaveShared_7,zoneWeld,toolWeldGun\WObj:=wobjCurrent\Track:=trackShared_6;
        RefreshDisp\Y\Z,peSeam23_6,posAOSeam23_6,pSeam23_6,pSeamFound3_1,pSeamFound3_2;
        RefreshDisp\X,peSeam23_6,posAOSeam23_6,pSeam23_6,pSeamFound4_1,pSeamFound4_2;
        ArcL pSeam23_6,speedWeld,seamShared,weldShared_7\Weave:=weaveShared_7,zoneWeld,toolWeldGun\WObj:=wobjCurrent\Track:=trackShared_6;
        RefreshDisp\X\Y\Z,peSeam23_7,posAOSeam23_7,pSeam23_7,pSeamFound4_1,pSeamFound4_2;
        ArcL pSeam23_7,speedWeld,seamShared,weldShared_2\Weave:=weaveShared_2,zoneWeld,toolWeldGun\WObj:=wobjCurrent\Track:=trackShared_2;
        RefreshDisp\X\Y\Z,peSeam23_8,posAOSeam23_8,pSeam23_8,pSeamFound4_1,pSeamFound4_2;
        ArcLEnd pSeam23_8,speedWeld,seamShared,weldShared_2\Weave:=weaveShared_2,fine,toolWeldGun\WObj:=wobjCurrent\Track:=trackShared_2;
        MoveL GetAproachTarget(pSeam23_8),speedAir,zoneAir,toolWeldGun\WObj:=wobjCurrent;
        PDispOff;

        MoveAbsJ [[-98.5025,-46.6432,9.398,108.84,-28.2844,-170],[-794.21,-510.359,374.549,9E+09,9E+09,9E+09]],speedAir,zoneAir,toolWeldGun\WObj:=wobjCurrent;

    UNDO
        PDispOff;
    ENDPROC

    LOCAL PROC Seam_25()
        MoveAbsJ [[-52.7557,-43.8883,36.8223,15.4091,-52.0967,115.276],[-737.076,502.617,361.603,9E+09,9E+09,9E+09]],speedAir,zoneAir,toolWeldGun\WObj:=wobjCurrent;

        RefreshDisp\X\Y\Z,peSeam25_1,posAOSeam25_1,pSeam25_1,pSeamFound1_1,pSeamFound1_2;
        MoveJ GetAproachTarget(pSeam25_1),speedAir,zoneAir,toolWeldGun\WObj:=wobjCurrent;
        ArcLStart pSeam25_1,speedAproach,seamShared,weldShared_1\Weave:=weaveShared_1,fine,toolWeldGun\WObj:=wobjCurrent\Track:=trackShared_1\SeamName:="WeldSeam";
        RefreshDisp\X\Y\Z,peSeam25_2,posAOSeam25_2,pSeam25_2,pSeamFound1_1,pSeamFound1_2;
        ArcL pSeam25_2,speedWeld,seamShared,weldShared_1\Weave:=weaveShared_1,zoneWeld,toolWeldGun\WObj:=wobjCurrent\Track:=trackShared_1;
        RefreshDisp\X\Y\Z,peSeam25_3,posAOSeam25_3,pSeam25_3,pSeamFound1_1,pSeamFound1_2;
        ArcL pSeam25_3,speedWeld,seamShared,weldShared_1\Weave:=weaveShared_1,zoneWeld,toolWeldGun\WObj:=wobjCurrent\Track:=trackShared_1;
        RefreshDisp\Y\Z,peSeam25_4,posAOSeam25_4,pSeam25_4,pSeamFound1_1,pSeamFound1_2;
        RefreshDisp\X,peSeam25_4,posAOSeam25_4,pSeam25_4,pSeamFound2_1,pSeamFound2_2;
        ArcL pSeam25_4,speedWeld,seamShared,weldShared_1\Weave:=weaveShared_1,zoneWeld,toolWeldGun\WObj:=wobjCurrent\Track:=trackShared_1;
        RefreshDisp\Y\Z,peSeam25_5,posAOSeam25_5,pSeam25_5,pSeamFound1_1,pSeamFound1_2;
        RefreshDisp\X,peSeam25_5,posAOSeam25_5,pSeam25_5,pSeamFound2_1,pSeamFound2_2;
        ArcL pSeam25_5,speedAproach,seamShared,weldShared_6\Weave:=weaveShared_6,zoneWeld,toolWeldGun\WObj:=wobjCurrent\Track:=trackShared_7;
        RefreshDisp\Y\Z,peSeam25_6,posAOSeam25_6,pSeam25_6,pSeamFound1_1,pSeamFound1_2;
        RefreshDisp\X,peSeam25_6,posAOSeam25_6,pSeam25_6,pSeamFound2_1,pSeamFound2_2;
        ArcL pSeam25_6,speedWeld,seamShared,weldShared_6\Weave:=weaveShared_6,zoneWeld,toolWeldGun\WObj:=wobjCurrent\Track:=trackShared_7;
        RefreshDisp\X\Y\Z,peSeam25_7,posAOSeam25_7,pSeam25_7,pSeamFound2_1,pSeamFound2_2;
        ArcL pSeam25_7,speedWeld,seamShared,weldShared_2\Weave:=weaveShared_2,zoneWeld,toolWeldGun\WObj:=wobjCurrent\Track:=trackShared_2;
        RefreshDisp\X\Y\Z,peSeam25_8,posAOSeam25_8,pSeam25_8,pSeamFound2_1,pSeamFound2_2;
        ArcLEnd pSeam25_8,speedWeld,seamShared,weldShared_2\Weave:=weaveShared_2,fine,toolWeldGun\WObj:=wobjCurrent\Track:=trackShared_2;
        MoveL GetAproachTarget(pSeam25_8),speedAir,zoneAir,toolWeldGun\WObj:=wobjCurrent;
        PDispOff;

        MoveAbsJ [[-94.6272,-62.3288,31.5236,-67.9884,-28.6289,132.373],[-732.484,502.809,100,9E+09,9E+09,9E+09]],speedAir,zoneAir,toolWeldGun\WObj:=wobjCurrent;

    UNDO
        PDispOff;
    ENDPROC

    LOCAL PROC Seam_27()
        MoveAbsJ [[-52.7557,-43.8883,36.8223,15.4091,-52.0967,115.276],[-737.076,502.617,361.603,9E+09,9E+09,9E+09]],speedAir,zoneAir,toolWeldGun\WObj:=wobjCurrent;

        RefreshDisp\X\Y\Z,peSeam27_1,posAOSeam27_1,pSeam27_1,pSeamFound1_1,pSeamFound1_2;
        MoveJ GetAproachTarget(pSeam27_1),speedAir,zoneAir,toolWeldGun\WObj:=wobjCurrent;
        ArcLStart pSeam27_1,speedAproach,seamShared,weldShared_1\Weave:=weaveShared_1,fine,toolWeldGun\WObj:=wobjCurrent\Track:=trackShared_1\SeamName:="WeldSeam";
        RefreshDisp\X\Y\Z,peSeam27_2,posAOSeam27_2,pSeam27_2,pSeamFound1_1,pSeamFound1_2;
        ArcL pSeam27_2,speedWeld,seamShared,weldShared_1\Weave:=weaveShared_1,zoneWeld,toolWeldGun\WObj:=wobjCurrent\Track:=trackShared_1;
        RefreshDisp\X\Y\Z,peSeam27_3,posAOSeam27_3,pSeam27_3,pSeamFound1_1,pSeamFound1_2;
        ArcL pSeam27_3,speedWeld,seamShared,weldShared_1\Weave:=weaveShared_1,zoneWeld,toolWeldGun\WObj:=wobjCurrent\Track:=trackShared_1;
        RefreshDisp\Y\Z,peSeam27_4,posAOSeam27_4,pSeam27_4,pSeamFound1_1,pSeamFound1_2;
        RefreshDisp\X,peSeam27_4,posAOSeam27_4,pSeam27_4,pSeamFound2_1,pSeamFound2_2;
        ArcL pSeam27_4,speedWeld,seamShared,weldShared_1\Weave:=weaveShared_1,zoneWeld,toolWeldGun\WObj:=wobjCurrent\Track:=trackShared_1;
        RefreshDisp\Y\Z,peSeam27_5,posAOSeam27_5,pSeam27_5,pSeamFound1_1,pSeamFound1_2;
        RefreshDisp\X,peSeam27_5,posAOSeam27_5,pSeam27_5,pSeamFound2_1,pSeamFound2_2;
        ArcL pSeam27_5,speedAproach,seamShared,weldShared_6\Weave:=weaveShared_6,zoneWeld,toolWeldGun\WObj:=wobjCurrent\Track:=trackShared_7;
        RefreshDisp\Y\Z,peSeam27_6,posAOSeam27_6,pSeam27_6,pSeamFound1_1,pSeamFound1_2;
        RefreshDisp\X,peSeam27_6,posAOSeam27_6,pSeam27_6,pSeamFound2_1,pSeamFound2_2;
        ArcL pSeam27_6,speedWeld,seamShared,weldShared_6\Weave:=weaveShared_6,zoneWeld,toolWeldGun\WObj:=wobjCurrent\Track:=trackShared_7;
        RefreshDisp\X\Y\Z,peSeam27_7,posAOSeam27_7,pSeam27_7,pSeamFound2_1,pSeamFound2_2;
        ArcL pSeam27_7,speedWeld,seamShared,weldShared_2\Weave:=weaveShared_2,zoneWeld,toolWeldGun\WObj:=wobjCurrent\Track:=trackShared_2;
        RefreshDisp\X\Y\Z,peSeam27_8,posAOSeam27_8,pSeam27_8,pSeamFound2_1,pSeamFound2_2;
        ArcLEnd pSeam27_8,speedWeld,seamShared,weldShared_2\Weave:=weaveShared_2,fine,toolWeldGun\WObj:=wobjCurrent\Track:=trackShared_2;
        MoveL GetAproachTarget(pSeam27_8),speedAir,zoneAir,toolWeldGun\WObj:=wobjCurrent;
        PDispOff;

        MoveAbsJ [[-94.6272,-62.3288,31.5236,-67.9884,-28.6289,132.373],[-732.484,502.809,100,9E+09,9E+09,9E+09]],speedAir,zoneAir,toolWeldGun\WObj:=wobjCurrent;

    UNDO
        PDispOff;
    ENDPROC

    LOCAL PROC Seam_26()
        MoveAbsJ [[-130.927,-60.2857,31.9214,-11.7127,-13.6227,-93.7947],[-632.831,-462.628,344.22,9E+09,9E+09,9E+09]],speedAir,zoneAir,toolWeldGun\WObj:=wobjCurrent;

        RefreshDisp\X\Y\Z,peSeam26_1,posAOSeam26_1,pSeam26_1,pSeamFound3_1,pSeamFound3_2;
        MoveJ GetAproachTarget(pSeam26_1),speedAir,zoneAir,toolWeldGun\WObj:=wobjCurrent;
        ArcLStart pSeam26_1,speedAproach,seamShared,weldShared_1\Weave:=weaveShared_1,fine,toolWeldGun\WObj:=wobjCurrent\Track:=trackShared_1\SeamName:="WeldSeam";
        RefreshDisp\X\Y\Z,peSeam26_2,posAOSeam26_2,pSeam26_2,pSeamFound3_1,pSeamFound3_2;
        ArcL pSeam26_2,speedWeld,seamShared,weldShared_1\Weave:=weaveShared_1,zoneWeld,toolWeldGun\WObj:=wobjCurrent\Track:=trackShared_1;
        RefreshDisp\X\Y\Z,peSeam26_3,posAOSeam26_3,pSeam26_3,pSeamFound3_1,pSeamFound3_2;
        ArcL pSeam26_3,speedWeld,seamShared,weldShared_1\Weave:=weaveShared_1,zoneWeld,toolWeldGun\WObj:=wobjCurrent\Track:=trackShared_1;
        RefreshDisp\Y\Z,peSeam26_4,posAOSeam26_4,pSeam26_4,pSeamFound3_1,pSeamFound3_2;
        RefreshDisp\X,peSeam26_4,posAOSeam26_4,pSeam26_4,pSeamFound4_1,pSeamFound4_2;
        ArcL pSeam26_4,speedWeld,seamShared,weldShared_1\Weave:=weaveShared_1,zoneWeld,toolWeldGun\WObj:=wobjCurrent\Track:=trackShared_1;
        RefreshDisp\Y\Z,peSeam26_5,posAOSeam26_5,pSeam26_5,pSeamFound3_1,pSeamFound3_2;
        RefreshDisp\X,peSeam26_5,posAOSeam26_5,pSeam26_5,pSeamFound4_1,pSeamFound4_2;
        ArcL pSeam26_5,speedAproach,seamShared,weldShared_7\Weave:=weaveShared_7,zoneWeld,toolWeldGun\WObj:=wobjCurrent\Track:=trackShared_6;
        RefreshDisp\Y\Z,peSeam26_6,posAOSeam26_6,pSeam26_6,pSeamFound3_1,pSeamFound3_2;
        RefreshDisp\X,peSeam26_6,posAOSeam26_6,pSeam26_6,pSeamFound4_1,pSeamFound4_2;
        ArcL pSeam26_6,speedWeld,seamShared,weldShared_7\Weave:=weaveShared_7,zoneWeld,toolWeldGun\WObj:=wobjCurrent\Track:=trackShared_6;
        RefreshDisp\X\Y\Z,peSeam26_7,posAOSeam26_7,pSeam26_7,pSeamFound4_1,pSeamFound4_2;
        ArcL pSeam26_7,speedWeld,seamShared,weldShared_2\Weave:=weaveShared_2,zoneWeld,toolWeldGun\WObj:=wobjCurrent\Track:=trackShared_2;
        RefreshDisp\X\Y\Z,peSeam26_8,posAOSeam26_8,pSeam26_8,pSeamFound4_1,pSeamFound4_2;
        ArcLEnd pSeam26_8,speedWeld,seamShared,weldShared_2\Weave:=weaveShared_2,fine,toolWeldGun\WObj:=wobjCurrent\Track:=trackShared_2;
        MoveL GetAproachTarget(pSeam26_8),speedAir,zoneAir,toolWeldGun\WObj:=wobjCurrent;
        PDispOff;

        MoveAbsJ [[-98.5025,-46.6432,9.398,108.84,-28.2844,-170],[-794.21,-510.359,374.549,9E+09,9E+09,9E+09]],speedAir,zoneAir,toolWeldGun\WObj:=wobjCurrent;

    UNDO
        PDispOff;
    ENDPROC

    LOCAL PROC Seam_28()
        MoveAbsJ [[-130.927,-60.2857,31.9214,-11.7127,-13.6227,-93.7947],[-632.831,-462.628,344.22,9E+09,9E+09,9E+09]],speedAir,zoneAir,toolWeldGun\WObj:=wobjCurrent;

        RefreshDisp\X\Y\Z,peSeam28_1,posAOSeam28_1,pSeam28_1,pSeamFound3_1,pSeamFound3_2;
        MoveJ GetAproachTarget(pSeam28_1),speedAir,zoneAir,toolWeldGun\WObj:=wobjCurrent;
        ArcLStart pSeam28_1,speedAproach,seamShared,weldShared_1\Weave:=weaveShared_1,fine,toolWeldGun\WObj:=wobjCurrent\Track:=trackShared_1\SeamName:="WeldSeam";
        RefreshDisp\X\Y\Z,peSeam28_2,posAOSeam28_2,pSeam28_2,pSeamFound3_1,pSeamFound3_2;
        ArcL pSeam28_2,speedWeld,seamShared,weldShared_1\Weave:=weaveShared_1,zoneWeld,toolWeldGun\WObj:=wobjCurrent\Track:=trackShared_1;
        RefreshDisp\X\Y\Z,peSeam28_3,posAOSeam28_3,pSeam28_3,pSeamFound3_1,pSeamFound3_2;
        ArcL pSeam28_3,speedWeld,seamShared,weldShared_1\Weave:=weaveShared_1,zoneWeld,toolWeldGun\WObj:=wobjCurrent\Track:=trackShared_1;
        RefreshDisp\Y\Z,peSeam28_4,posAOSeam28_4,pSeam28_4,pSeamFound3_1,pSeamFound3_2;
        RefreshDisp\X,peSeam28_4,posAOSeam28_4,pSeam28_4,pSeamFound4_1,pSeamFound4_2;
        ArcL pSeam28_4,speedWeld,seamShared,weldShared_1\Weave:=weaveShared_1,zoneWeld,toolWeldGun\WObj:=wobjCurrent\Track:=trackShared_1;
        RefreshDisp\Y\Z,peSeam28_5,posAOSeam28_5,pSeam28_5,pSeamFound3_1,pSeamFound3_2;
        RefreshDisp\X,peSeam28_5,posAOSeam28_5,pSeam28_5,pSeamFound4_1,pSeamFound4_2;
        ArcL pSeam28_5,speedAproach,seamShared,weldShared_7\Weave:=weaveShared_7,zoneWeld,toolWeldGun\WObj:=wobjCurrent\Track:=trackShared_6;
        RefreshDisp\Y\Z,peSeam28_6,posAOSeam28_6,pSeam28_6,pSeamFound3_1,pSeamFound3_2;
        RefreshDisp\X,peSeam28_6,posAOSeam28_6,pSeam28_6,pSeamFound4_1,pSeamFound4_2;
        ArcL pSeam28_6,speedWeld,seamShared,weldShared_7\Weave:=weaveShared_7,zoneWeld,toolWeldGun\WObj:=wobjCurrent\Track:=trackShared_6;
        RefreshDisp\X\Y\Z,peSeam28_7,posAOSeam28_7,pSeam28_7,pSeamFound4_1,pSeamFound4_2;
        ArcL pSeam28_7,speedWeld,seamShared,weldShared_2\Weave:=weaveShared_2,zoneWeld,toolWeldGun\WObj:=wobjCurrent\Track:=trackShared_2;
        RefreshDisp\X\Y\Z,peSeam28_8,posAOSeam28_8,pSeam28_8,pSeamFound4_1,pSeamFound4_2;
        ArcLEnd pSeam28_8,speedWeld,seamShared,weldShared_2\Weave:=weaveShared_2,fine,toolWeldGun\WObj:=wobjCurrent\Track:=trackShared_2;
        MoveL GetAproachTarget(pSeam28_8),speedAir,zoneAir,toolWeldGun\WObj:=wobjCurrent;
        PDispOff;

        MoveAbsJ [[-98.5025,-46.6432,9.398,108.84,-28.2844,-170],[-794.21,-510.359,374.549,9E+09,9E+09,9E+09]],speedAir,zoneAir,toolWeldGun\WObj:=wobjCurrent;

    UNDO
        PDispOff;
    ENDPROC

ENDMODULE
